      U     #S1; // Select No. 1
      SPB   S1;
      U     #S2; // Select No. 2
      SPB   S2;
      U     #S3; // Select No. 3
      SPB   S3;
      U     #S4; // Select No. 4
      SPB   S4;
      SPA   OFF;

S1:   L     P##ANY1; // Load the Pointer of ANY 1
      L     1; // Wert für Kanalanzeige
      SPA   SAVE;
S2:   L     P##ANY2; // Load the Pointer of ANY 2
      L     2;
      SPA   SAVE;
S3:   L     P##ANY3; // Load the Pointer of ANY 3
      L     3;
      SPA   SAVE;
S4:   L     P##ANY4; // Load the Pointer of ANY 4
      L     4;
      SPA   SAVE;

OFF:  L     P##anyNull; // Create a temporary
      LAR1  ; // NullAny
      L     DW#16#0;
      T     D [AR1,P#0.0];
      T     D [AR1,P#4.0];
      T     W [AR1,P#8.0];

      L     P##anyNull; // Load Pointer to temporary NullAny
      L     0;
      CLR   ; // CLR BIE

SAVE: SAVE  ; // FC-ENO: TRUE IF ChannelSelected
      T     #DSP_CHANNEL; // Anzeige aktiver Kanal
      TAK   ; // P##ANY in AKKU1 zurück
      LAR1  ; // Load the Pointer of the Source Any into AR1
      L     P##RET_VAL; // Load the Pointer of the ReturnValue into
      LAR2  ; // AR2

      L     D [AR1,P#0.0]; // Copy the 10 Bytes of the ANY Pointer to
      T     D [AR2,P#0.0]; // the returned ANY

      L     D [AR1,P#4.0];
      T     D [AR2,P#4.0];

      L     W [AR1,P#8.0];
      T     W [AR2,P#8.0];


END_FUNCTION

FUNCTION "m7b_DB_COMPARE_ByRef" : VOID
TITLE =DB_COMPARE_ByRef
//Vergleicht Anzahl Bytes von 2 Datenbausteinen
//Die Vergleichsroutine arbeitet sehr effektiv, da die Werte nicht als 8-Bit
//sondern als 32-Bit-Werte verglichen werden. Weiterhin müssen die DBs nur einmal
//geöffnet werden, dies erreicht man, indem man einen DB als Global-DB und den
//anderen als Instanz-DB öffnet.
//
//AUTOR: Stefan Maag, Dipl.-Ing. (FH) Elektrotechnik
//DATUM: 10/2010
//INTERNET: www.maagic7.de
//
//AENDERUNGSVERMERKE:
//--------------------------------------------------------------------------------
//DATUM        NAME        AENDERUNG
//--------------------------------------------------------------------------------
//19.10.2010   S.Maag      Basiert auf FC2 CopyDBW_ByRef
//25.10.2010   S.Maag      Wenn keine Einzelbytes mehr zu kopieren sind, dann
//                         darf man nicht zu END springen sondern zu EQ (Daten
//                         gleich)
//--------------------------------------------------------------------------------
//
//HINWEISE:
AUTHOR : 'S.Maag'
FAMILY : Maagic7
VERSION : 0.1


VAR_INPUT
  SOURCE : BLOCK_DB ;
  DEST : BLOCK_DB ;
  SOURCE_BYTE : INT ;
  DEST_Byte : INT ;
  NoOfBytes : INT ;
END_VAR
VAR_TEMP
  QUELL_ADR : DINT ;
  ZIEL_ADR : DINT ;
  AR1 : DINT ;
  LOOPS : INT ;
END_VAR
BEGIN
NETWORK
TITLE =Register sichern
//Adressregister 2 Global- und Instanz DB werden bei CALL-Aufrufen automatisch
//vom System gesichert, bei UC nicht!
      TAR1  #AR1; // Adressregister 1 sichern

NETWORK
TITLE =Adressen für Quell und Ziel-DW als Pointer in Adressregister

      L     #SOURCE_BYTE; // Quelldatenbyte Nr.
      SLD   3; // als Pointer
      L     P#0.0; // 0-Pointer addieren, damit
      +D    ; // Kennungsbits für Pointer gesetzt werden
      LAR1  ; // ins Adressregister 1

      L     #DEST_Byte; // ZieldatenByte-Nr
      SLD   3; // als Pointer
      L     P#0.0;
      +D    ;
      LAR2  ; // ins Adressregister 2
NETWORK
TITLE =Daten vergleichen

      AUF   #SOURCE; // Quell-DB als Global-DB öffnen
      TDB   ; // Global und Instanz-DB tauschen (Quelle wird Instanz-DB)
      AUF   #DEST; // Ziel-DB als Global-DB öffnen

      L     #NoOfBytes; // Anzahl der zu kopierenden Bytes
      L     4; // in Anzahl der 32-Bit-Werte umrechen
      /I    ;
      SPZ   LAST; // Wenn 0 32-Bit Werte, dann weiter mit letzten 3 Bytes
LOOP: T     #LOOPS;
      L     DID [AR1,P#0.0]; // QuellDaten lesen
      L     DBD [AR2,P#0.0]; // VergleichsDaten lesen
      <>D   ; // wenn nicht gleich, dann Ende
      SPB   NEQ;
      +AR1  P#4.0; // Quell-Pointer in AR1 um 4 Bytes erhöhen
      +AR2  P#4.0; // Ziel-Pointer in AR2 um 4 Bytes erhöhen
      L     #LOOPS; // Schleifenzähler wieder in Akku 1 zurück
      LOOP  LOOP; // Schleifenzähler bearbeiten

LAST: L     #NoOfBytes; // nun noch die evtl. letzte 3 Bytes prüfen
      L     2#11; // Anzahl übriger Bytes maskieren
      UW    ; // Anzahl übriger Bytes
      SPZ   EQ; // Wenn 0 dann ENDE
LOP1: T     #LOOPS;
      L     DIB [AR1,P#0.0]; // QuellDaten lesen
      L     DBB [AR2,P#0.0]; // VergleichsDaten lesen
      <>I   ; // wenn nicht gleich, dann Ende
      SPB   NEQ;
      +AR1  P#1.0; // Quell-Pointer in AR1 um 1 Byte erhöhen
      +AR2  P#1.0; // Vergleichs-Pointer in AR2 um 1 Byte erhöhen
      L     #LOOPS; // Schleifenzähler wieder in Akku 1 zurück
      LOOP  LOP1; // Schleifenzähler bearbeiten

EQ:   SET   ; // Daten sind gleich  (equal)
      SAVE  ; // ENO=TRUE
      CLR   ;
      SPA   END;

NEQ:  CLR   ; // Daten sind nicht identisch (not equal)
      SAVE  ; // ENO=FALSE

NETWORK
TITLE =Adressregister 1 wieder herstellen

END:  LAR1  #AR1; // Adressregister 1 wieder herstellen

END_FUNCTION

FUNCTION "m7b_IEC_TIMER_CTRL" : VOID
TITLE =Erweiterte Steuerung von IEC Timern (RESET und 0ms Rüfung)
//IEC-Timer haben im Gegensatz zu den S5-Timern keine RESET-Eingang
//Für RESET eines IEC-Timers muss man diesen mit einer Zeit von 0ms
//aufrufen. (Dies gilt dann als Reset). D.h. IEC-Timer laufen mit
//einer Vorgabe von 0ms nicht an. S5-Timer dagegen gehen bei 0s sofort auf Hi.
//Dieses Verhalten der IEC-Timer führt immer wieder zu Problemen, wenn variable
//Zeitwerte verwendet werden, und 0 eingegeben wird.
//
//Dieser Baustein vor den eigentlichen IEC-Timer geschaltet, ermöglicht gleiches
//Verhalten wie bei S5-Timern.
//
//AUTOR: Stefan Maag, Dipl.-Ing. (FH) Elektrotechnik
//DATUM: 1/2013
//INTERNET: www.maagic7.de
//
//AENDERUNGSVERMERKE:
//--------------------------------------------------------------------------------
//DATUM        NAME        AENDERUNG
//--------------------------------------------------------------------------------
//
//--------------------------------------------------------------------------------
//
//HINWEISE:
AUTHOR : 'S.Maag'
FAMILY : Maagic7
VERSION : 0.1


VAR_INPUT
  IN_TIME : TIME ;	//Vorgabezeit Timer
  RESET : BOOL ;	//RESET Timer
END_VAR
VAR_OUTPUT
  OUT_TIME : TIME ;
END_VAR
BEGIN
NETWORK
TITLE =

      SET   ;
      SAVE  ;
      CLR   ;

NETWORK
TITLE =

      L     T#0MS; // Wenn Reset, dann 0ms als Zeit ausgeben
      U     #RESET; // Ein Aufruf mit T=0ms ist für IEC Timer
      SPB   save; // Ein Reset. Siehe Step7 Dokumentation

      L     T#1MS; // Wenn kein Reset, dann minimale Zeitvorgabe
      L     #IN_TIME; // auf 1ms begrenzen
      <D    ; // sonst läuft Timer nicht los,
      SPB   save; // d.h. Ausgang bleibt Lo, da RESET
      TAK   ;
save: T     #OUT_TIME; // Ausgang Zeit für IEC-Timer

END_FUNCTION

FUNCTION "m7b_IEC_TIMER_WRAPPER" : VOID
TITLE =IEC-TIMER-WRAPPER
//AUTOR: Stefan Maag, Dipl.-Ing. (FH) Elektrotechnik
//DATUM: 8/2013
//INTERNET: www.maagic7.de
//
//AENDERUNGSVERMERKE:
//--------------------------------------------------------------------------------
//DATUM        NAME            AENDERUNG
//--------------------------------------------------------------------------------
//
//--------------------------------------------------------------------------------
//
//HINWEISE:
AUTHOR : 'S.Maag'
FAMILY : Maagic7
VERSION : 0.1


VAR_INPUT
  IN : BOOL ;	//TIMER IN-SIGNAL
  RESET : BOOL ;	//RESET THE TIMER
  cfgDSP_ET_INV : BOOL ;	//Configuration: Display the ET-Time inverted (rest TIME)
  PT : TIME ;	//TIMER PT (TIME)
  ptrTmrInst : POINTER ;	//RELATIVE POINTER TO TIMER INSTANCE: MemoryArea must be in actual instance DB
  TMR_SFB_No : INT ;	//No. of Timer SFB: 3=TP, 4=TON, 5=TOF
END_VAR
VAR_OUTPUT
  ET : TIME ;	//Abgelaufene Zeit
END_VAR
VAR_TEMP
  memAR1 : DWORD ;
  memAR2 : DWORD ;
  TimeIsNull : BOOL ;
END_VAR
BEGIN
NETWORK
TITLE =Save AR1 & AR2

      TAR1  #memAR1; // save AR1, AR2
      TAR2  #memAR2;

NETWORK
TITLE =Load AR2 with Pointer to TIMER-INSTANCE and SET the TIMER
//For the unconditioned call of TIMER SFBs (UC SFB3..5) we have to implement the
//following steps manually:
//1. SET AR2 with correct INSTANCE-POINTER of TIMER
//2. TRANSFER TIMER.VARIABLES into INCTANCE-DATA: (IN and PT)
//
//TIMER_STRUCTURE of SFB 3..5 (TP/TON/TOF) with relative ADDRESS
//   IN      BOOL   0.0  INPUT:  Signal
//   PT      TIME   2.0  INPUT:  TIME
//   Q       BOOL   6.0  OUTPUT: Q
//   ET      TIME   8.0  OUTPUT: ET
//   STATE   BYTE  10.0  static: STATE
//   STIME   TIME  14.0  static: STIME
//   ATIME   TIME  18.0  static: ATIME
//
      L     P##ptrTmrInst; // Load POINTER to ptrTmrInst
      LAR1  ; // in AR1
      L     D [AR1,P#2.0]; // Load relative InstancePointer (Offset 2: don't need DB-No; Byte 0..1)
      UD    DW#16#FFFFFF; // BYTE.BIT-Pointer only: Remove MemoryArea (Speicherbereich)
      +AR2  ; // Instance-DataPointer of TimerInstance [P#Byte.Bit]
      U     #IN; // Timer Startsignal in Instanz eintragen
      =     DIX [AR2,P#0.0]; // [TIMER].IN

      L     #PT; // Zeitwert in TimerInstanz eintragen
      T     DID [AR2,P#2.0]; // [TIMER].PT
      L     L#0; // IF .PT =0 means RESET for IEC-TIMERs
      ==D   ;
      =     #TimeIsNull; // Zeit ist T#0ms  => [TIMER].Q will be FALSE

NETWORK
TITLE =RESET
//// IEC-Timer Reset is done by PT:=0
//IF RESET THEN
//   [TIMER].PT = 0
//ENDIF
      U     #RESET;
      SPBN  ne2;
      L     L#0; // T#0ms means RESET for IEC-TIMERs
      T     DID [AR2,P#2.0]; // [TIMER].PT

ne2:  NOP   0;
NETWORK
TITLE =SELECT TIMER FUNCTION
//SELECT TMR_SFB_No
//  CASE <3 or >5 : ERR
//  CASE 3: SFB3 'TP'
//  CASE 4: SFB4 'TON'
//  CASE 5: SFB5 'TOF'
      L     #TMR_SFB_No;
      SPL   ERR; // >5 (OUT OF RANGE)
      SPA   ERR; // 0
      SPA   ERR; // 1
      SPA   ERR; // 2
      SPA   TP; // 3  SFB3 TP
      SPA   TON; // 4  SFB4 TON
      SPA   TOF; // 5  SFB5 TOF

ERR:  NOP   0; //  *****    E R O R     *****
      CLR   ;
      SAVE  ;
      SPA   END;

TP:   NOP   0; //  ***** M O D E   T P  *****

      UC    "TP"; // unconditioned call for SFB3 'TP'; AR2 has to be loaded with InstanceDataPointer first!

      U     DIX [AR2,P#6.0]; // [TIMER].Q
      SAVE  ;
      CLR   ;
      SPA   END;

TON:  NOP   0; // ***** M O D E   T O N *****

      UC    "TON"; // unconditioned call for SFB4 'TON'; AR2 has to be loaded with InstanceDataPointer first!

      U     #IN; // INPUT SIGNAL for TIMER start
      U     #TimeIsNull;
      O     DIX [AR2,P#6.0]; // [TIMER].Q
      SAVE  ;
      CLR   ;
      SPA   END;

TOF:  NOP   0; // ***** M O D E   T O F *****

      UC    "TOF"; // unconditioned call for SFB5 'TOF'; AR2 has to be loaded with InstanceDataPointer first!

      U     #IN; // INPUT SIGNAL for TIMER start
      U     #TimeIsNull;
      O     DIX [AR2,P#6.0]; // [TIMER].Q
      SAVE  ;
      CLR   ;
      SPA   END;


END:  L     DID [AR2,P#8.0]; // [TIMER].ET   (Laufzeit vom IEC-Timer)
      UN    #cfgDSP_ET_INV; // config Input: Display Time inverted (RestZeit)
      SPB   save;
      L     #PT; // IF inverted THEN
      TAK   ; //    [OUT].ET = PT-TIMER.ET
      -D    ;
save: T     #ET; // [OUT].ET

      LAR1  #memAR1; // restore AR1, AR2
      LAR2  #memAR2;


END_FUNCTION

FUNCTION "m7b_InputControl_REAL" : VOID
TITLE =Input Control for REAL
//Eingabekontrolle für REAL-Werte.
//Begrenzt einen Real-Wert auf vorgegebenen Min/Max Grenzen,
//wobei die Begrenzungsfunktion über Konfigurationseingänge
//zu und abgeschaltet werden kann. So lassen sich z.B. über globale
//Schalter die Eingabebegrenzungen z.B. für Servicezwecke aufheben.
//
//[IN]
//rMIN :         Zulässiger Minimalwert
//rMAX :         Zulässiger Maximalwert
//cfg_LIM_min :  Konfiguration Begrenzung auf Min-Wert aktiv
//cfg_LIM_max :  Konfiguration Begrenzung auf Max-Wert aktiv
//
//[INOUT]
//rVALUE :       Zu prüfender/begrenzender Wert
//
//[OUT]
//MSG_LIM_MAX :  Meldung: Max-Limit überschritten
//MSG_LIM_MIN :  Meldung: Min-Limit unterschritten
//DSP_STATUS :   Status: 0 : o.k. ; 1 : MinLimit; 2 : MaxLimit
//
//AUTOR: Stefan Maag, Dipl.-Ing. (FH) Elektrotechnik
//DATUM: 5/2013
//INTERNET: www.maagic7.de
//
//AENDERUNGSVERMERKE:
//--------------------------------------------------------------------------------
//DATUM        NAME            AENDERUNG
//--------------------------------------------------------------------------------
//
//--------------------------------------------------------------------------------
//
//HINWEISE:
AUTHOR : 'S.Maag'
FAMILY : Maagic7
VERSION : 0.1


VAR_INPUT
  rMIN : REAL ;	//Zulässiger Minimalwert
  rMAX : REAL ;	//Zulässiger Maximalwert
  cfg_LIM_min : BOOL ;	//Konfiguration Begrenzung auf Min-Wert aktiv
  cfg_LIM_max : BOOL ;	//Konfiguration Begrenzung auf Max-Wert aktiv
END_VAR
VAR_OUTPUT
  MSG_LIM_MAX : BOOL ;	//Meldung: Max-Limit überschritten
  MSG_LIM_MIN : BOOL ;	//Meldung: Min-Limit unterschritten
  DSP_STATUS : INT ;	//Status: 0 : o.k. ; 1 : MinLimit; 2 : MaxLimit
END_VAR
VAR_IN_OUT
  rVALUE : REAL ;	//Zu prüfender Wert
END_VAR
BEGIN
NETWORK
TITLE =
//-
      SET   ;
      SAVE  ;
      CLR   ;
NETWORK
TITLE =Begrenzung, wenn aktiv!
//Begrenzen des Wertes, wenn über-/unterschritten
//Begrenzung wird mit den Konfigurationseingängen
//cfg_LIM_min, cfg_LIM_max = HIGH aktiviert.
      L     #rVALUE; // Sollwert
      L     #rMIN; // minimal Wert
      <R    ;
      U     #cfg_LIM_min;
      SPB   LIM; // Limitierung wenn VALUE < MIN
      TAK   ; // VALUE wieder in Akku 1
      L     #rMAX; // Maximalwert
      >R    ;
      U     #cfg_LIM_max;
      SPB   LIM; // Limitierung wenn VALUE > MAX

      SPA   ne;
      CLR   ; // VKE löschen, da keine Begrenzung erfolgte
      SAVE  ; // BIE-Bit = 0, da Wert im Bereich war; ="Keine Begrenzung"
      BEA   ;

LIM:  T     #rVALUE; // max.Wert als Sollwert ausgeben

ne:   NOP   0;

NETWORK
TITLE =Meldeausgänge Limit überschritten
//-
      L     #rVALUE;
      L     #rMAX; // minmal zulässiger Wert
      >R    ; // falls MIN > VALUE
      =     #MSG_LIM_MAX;

      L     #rVALUE;
      L     #rMIN; // minmal zulässiger Wert
      <R    ; // falls MIN > VALUE
      =     #MSG_LIM_MIN;

NETWORK
TITLE =STATUS
//0 : o.k., keine Begreunzung aktiv
//1 : Begrenzung min
//2 : Begrenzung max
      L     1;
      U     #MSG_LIM_MIN;
      SPB   save;

      L     2;
      U     #MSG_LIM_MAX;
      SPB   save;

      L     0;
save: T     #DSP_STATUS;
END_FUNCTION

FUNCTION "m7b_InputControl_DINT" : VOID
TITLE =Input Control for DINT
//Eingabekontrolle für DINT-Werte.
//Begrenzt einen Real-Wert auf vorgegebenen Min/Max Grenzen,
//wobei die Begrenzungsfunktion über Konfigurationseingänge
//zu und abgeschaltet werden kann. So lassen sich z.B. über globale
//Schalter die Eingabebegrenzungen z.B. für Servicezwecke aufheben.
//
//[IN]
//dMIN :         Zulässiger Minimalwert
//dMAX :         Zulässiger Maximalwert
//cfg_LIM_min :  Konfiguration Begrenzung auf Min-Wert aktiv
//cfg_LIM_max :  Konfiguration Begrenzung auf Max-Wert aktiv
//
//[INOUT]
//dVALUE :       Zu prüfender/begrenzender Wert
//
//[OUT]
//MSG_LIM_MAX :  Meldung: Max-Limit überschritten
//MSG_LIM_MIN :  Meldung: Min-Limit unterschritten
//DSP_STATUS :   Status: 0 : o.k. ; 1 : MinLimit; 2 : MaxLimit
//
//AUTOR: Stefan Maag, Dipl.-Ing. (FH) Elektrotechnik
//DATUM: 10/2017
//INTERNET: www.maagic7.de
//
//AENDERUNGSVERMERKE:
//--------------------------------------------------------------------------------
//DATUM        NAME            AENDERUNG
//--------------------------------------------------------------------------------
//31.10.2017   S.Maag         Entstand aus FC252 InputControl_REAL
//--------------------------------------------------------------------------------
//
//HINWEISE:
AUTHOR : 'S.Maag'
FAMILY : Maagic7
VERSION : 0.1


VAR_INPUT
  dMIN : DINT ;	//Zulässiger Minimalwert
  dMAX : DINT ;	//Zulässiger Maximalwert
  cfg_LIM_min : BOOL ;	//Konfiguration Begrenzung auf Min-Wert aktiv
  cfg_LIM_max : BOOL ;	//Konfiguration Begrenzung auf Max-Wert aktiv
END_VAR
VAR_OUTPUT
  MSG_LIM_MAX : BOOL ;	//Meldung: Max-Limit überschritten
  MSG_LIM_MIN : BOOL ;	//Meldung: Min-Limit unterschritten
  DSP_STATUS : INT ;	//Status: 0 : o.k. ; 1 : MinLimit; 2 : MaxLimit
END_VAR
VAR_IN_OUT
  dVALUE : DINT ;	//Zu prüfender Wert
END_VAR
BEGIN
NETWORK
TITLE =
//-
      SET   ;
      SAVE  ;
      CLR   ;
NETWORK
TITLE =Begrenzung, wenn aktiv!
//Begrenzen des Wertes, wenn über-/unterschritten
//Begrenzung wird mit den Konfigurationseingängen
//cfg_LIM_min, cfg_LIM_max = HIGH aktiviert.
      L     #dVALUE; // Sollwert
      L     #dMIN; // minimal Wert
      <D    ;
      U     #cfg_LIM_min;
      SPB   LIM; // Limitierung wenn VALUE < MIN
      TAK   ; // VALUE wieder in Akku 1
      L     #dMAX; // Maximalwert
      >D    ;
      U     #cfg_LIM_max;
      SPB   LIM; // Limitierung wenn VALUE > MAX

      SPA   ne;
      CLR   ; // VKE löschen, da keine Begrenzung erfolgte
      SAVE  ; // BIE-Bit = 0, da Wert im Bereich war; ="Keine Begrenzung"
      BEA   ;

LIM:  T     #dVALUE; // max.Wert als Sollwert ausgeben

ne:   NOP   0;

NETWORK
TITLE =Meldeausgänge Limit überschritten
//-
      L     #dVALUE;
      L     #dMAX; // minmal zulässiger Wert
      >D    ; // falls MIN > VALUE
      =     #MSG_LIM_MAX;

      L     #dVALUE;
      L     #dMIN; // minmal zulässiger Wert
      <D    ; // falls MIN > VALUE
      =     #MSG_LIM_MIN;

NETWORK
TITLE =STATUS
//0 : o.k., keine Begreunzung aktiv
//1 : Begrenzung min
//2 : Begrenzung max
      L     1;
      U     #MSG_LIM_MIN;
      SPB   save;

      L     2;
      U     #MSG_LIM_MAX;
      SPB   save;

      L     0;
save: T     #DSP_STATUS;
END_FUNCTION

FUNCTION "m7b_BetriebsStunden" : VOID
TITLE =Betriebsstunden erfassen
//pro Bausteinaufruf wird eine bestimmte Anzahl von Sekunden addiert.
//Diesen Baustein mit einem Referenztakt (Timer OB, oder Flanke von Taktmerker
//aufrufen)
//
//AUTOR: Stefan Maag, Dipl.-Ing. (FH) Elektrotechnik
//DATUM: 8/2013
//INTERNET: www.maagic7.de
//
//AENDERUNGSVERMERKE:
//--------------------------------------------------------------------------------
//DATUM        NAME            AENDERUNG
//--------------------------------------------------------------------------------
//04.12.2013   S.Maag      Bei Count-Aufruf über EN, funktionieren Impulsausgänge
//                         nicht, deswegen Count-Eingang eingeführt
//--------------------------------------------------------------------------------
//
//HINWEISE:
AUTHOR : 'S.Maag'
FAMILY : Maagic7
VERSION : 0.1


VAR_INPUT
  COUNT : BOOL ;	//Eingang zählen
  RESET : BOOL ;	//Tageszähler löschen
  SEC_ADD : INT ;
END_VAR
VAR_OUTPUT
  IMP_MIN : BOOL ;
  IMP_H : BOOL ;
END_VAR
VAR_IN_OUT
  sec : INT ;
  min : INT ;
  h : DINT ;	//Stunden
END_VAR
BEGIN
NETWORK
TITLE =

      SET   ;
      SAVE  ;
      R     #IMP_MIN;
      R     #IMP_H;
      CLR   ;

      UN    #RESET;
      SPB   cnt;
      L     0;
      T     #sec;
      T     #min;
      T     #h;
      BEA   ;

cnt:  UN    #COUNT;
      BEB   ;

      L     #sec;
      L     #SEC_ADD;
      +I    ;
      T     #sec;
      L     60;
      <I    ;
      BEB   ;

      S     #IMP_MIN;

      L     #sec;
      +     -60;
      T     #sec;

      L     #min;
      +     1;
      T     #min;

      L     60;
      <I    ;
      BEB   ;

      S     #IMP_H;

      L     #min;
      +     -60;
      T     #min;

      L     #h;
      +     1;
      T     #h;
      L     0; // Überlauf prüfen, Stunden müssen >=0 sein
      >=D   ; // wenn nicht, dann auf 0 setzten
      BEB   ;
      T     #h;
END_FUNCTION

FUNCTION "m7b_DeltaTime" : VOID
TITLE =DeltaTime : Zeitdifferenz zwischen 2 Impulsen
//Ermittelt den Abstand zwischen 2 Impulsen.
//In io_DeltaTime wird der Abstand des letzten Impulses gespeichert.
//DSP_ActTimDiff zeigt die seit letztem Impuls aktuell vergangene Zeit
//MAX_timDiff = MAX(io_DeltaTime, DSP_TimeDiffAkt)
//
//
//AUTOR: Stefan Maag, Dipl.-Ing. (FH) Elektrotechnik
//DATUM: 11/2013
//INTERNET: www.maagic7.de
//
//AENDERUNGSVERMERKE:
//--------------------------------------------------------------------------------
//DATUM        NAME        AENDERUNG
//--------------------------------------------------------------------------------
//04/09/2017   S.Maag      RESET Eingang + einfrieren 1sec vor max Differenz
//
//16/01/2014   S.Maag      ENO=TRUE
//
//03/12/2013   S.Maag      SFC64 TimeTick Zeitdifferenz korrigiert
//                         da 31Bit, Fehler bei Überlauf.
//                         jetzt Differenzber. mit FC256 "ABS_DIFF_S7SysTime"
//--------------------------------------------------------------------------------
//
//HINWEISE:
AUTHOR : 'S.Maag'
FAMILY : Maagic7
VERSION : 0.1


VAR_INPUT
  FP_Signal : BOOL ;	//Flanke Signal
  RESET : BOOL ;
END_VAR
VAR_OUTPUT
  DSP_ActTimeDiff : TIME ;	//Anzeige aktuelle Zeitdifferenz seit letztem Ereignis
  MAX_timDiff : TIME ;	//Max(timDiff, io_DeltaTime)
END_VAR
VAR_IN_OUT
  memTime : TIME ;
  io_DeltaTime : TIME ;
END_VAR
VAR_TEMP
  SysTimer : TIME ;
END_VAR
BEGIN
NETWORK
TITLE =

      SET   ;
      SAVE  ;
      CLR   ;

NETWORK
TITLE =
//31Bit = 7F FF FF FF = 2147483647 - 1000ms = 2147482647 ms
//1sec vor Ablauf der max Differenz den Differenzwert einfrieren bis neuer Impuls
//kommt.
//Dies verhindert Überlauf der Zeitdifferenz uns somit eine Rückfall der
//Differenzzeit auf 0 ohne neuen Impuls
      UN    #RESET;
      SPB   do;

      L     T#0MS;
      T     #DSP_ActTimeDiff;
      T     #MAX_timDiff;
      SPA   ne2;

do:   NOP   0;
      CALL "TIME_TCK" (
           RET_VAL                  := #SysTimer);

      L     #DSP_ActTimeDiff; // Wenn max. Zeitdifferenz erreicht,
      L     L#2147482647; // dann Wert einfrieren und erst
      >=D   ; // nach neuem Impuls weiter
      SPB   ne2; // dadurch wird ein überlauf verhindert

      L     #SysTimer;
      L     #memTime;
      UC    "m7b_ABS_DIFF_S7SysTime"; // Absolute Zeitdifferenz S7-SystemTimer 31Bit
      T     #DSP_ActTimeDiff;
      L     #io_DeltaTime;
      UC    FC    21;
      T     #MAX_timDiff;
ne2:  NOP   0;
NETWORK
TITLE =Zeit Ereignis

      UN    #FP_Signal;
      SPB   ne3;

      L     #DSP_ActTimeDiff;
      T     #io_DeltaTime;

      L     L#0;
      T     #DSP_ActTimeDiff;

      L     #SysTimer;
      T     #memTime;

ne3:  NOP   0;
NETWORK
TITLE =



END_FUNCTION

FUNCTION "m7b_CNT_UpDwn_IMP_MM.SS" : VOID
TITLE =Zählt Impulse im Minuten.Sekunden Format (MM.SS) - DINT
//Bei jedem Aufruf Zählt diese Funktion einen Impuls weiter. Die Wertedarstellung
//erfolgt im Minuten.Sekunden-Format MM.SS. Es wird also alle 60 Impulse ein
//Überlauf auf MM erzeugt. Dieser Baustein eignet sich zum Erfassen von z.B.
//Behälter Füll- und Entleerzeiten, wenn er mit einer Sekundenflanke aufgerufen
//wird. Am besten Flanke des Systemtaktmerkers 1 sec verwenden.
//
//Der FC-ENO Ausgang ist immer dan HIGH, wenn Zeit > 0
//
//AUTOR: Stefan Maag, Dipl.-Ing. (FH) Elektrotechnik
//DATUM: 5/2005
//
//AENDERUNGSVERMERKE:
//--------------------------------------------------------------------------------
//DATUM        NAME            AENDERUNG
//--------------------------------------------------------------------------------
//25.06.2019   S.Maag     COUNT_UP / COUNT_DOWN
//                        Ausgang d_mmss als I/O, somit muss nur bei Änderung
//                        neu berechnet werden.
//                        ENO = (Time > 0) d.h. ENO=FALSE, wenn Zeit = 0
//                        Wird für Rückwärtszählung benötigt!
//
//14.08.2013   S.Maag     Ausgang MM.SS hinzugefügt so dass im IO mem_dIMP die
//                        gezählten Impulse stehen und nicht mehr MM.SS
//--------------------------------------------------------------------------------
//
//HINWEISE:
AUTHOR : 'S.Maag'
FAMILY : Maagic7
VERSION : 0.1


VAR_INPUT
  COUNT_UP : BOOL ;	//Signal for counting up
  COUNT_DWN : BOOL ;	//Signal for counting down
  SET : BOOL ;	//Set to VALUE_SET
  VALUE_SET_mmss : DINT ;	//Value [mm:ss] to set
END_VAR
VAR_IN_OUT
  io_dIMP : DINT ;	//Memory for impulses [sec]
  io_d_mmss : DINT ;	//Memory [mm:ss] format
END_VAR
VAR_TEMP
  SS : INT ;
  MM : DINT ;
END_VAR
BEGIN
NETWORK
TITLE =



NETWORK
TITLE =SET

      UN    #SET;
      SPB   NE1;

      L     #VALUE_SET_mmss;
      L     L#100;
      MOD   ; // Sekundenanteil 0..99
      T     #SS; // =Divisionsrest = Sekunden

      L     #VALUE_SET_mmss;
      L     L#100; // Minutenanteil
      /D    ;
      T     #MM; // Rückrechnung auf Sekunden
      L     L#60; // damit werden automatisch
      *D    ; // Sekundenanteile von 60..99
      L     #SS; // auf eine zusätzliche Minute
      +D    ; // umgerechnet
      T     #io_dIMP;
      SPA   END;
NE1:  NOP   0;
NETWORK
TITLE =Impulse Zählen [mm:ss]
//
//
      U     #COUNT_UP;
      SPB   up;
      U     #COUNT_DWN;
      SPB   dwn;

      SPA   END;

up:   L     #io_dIMP;
      +     L#1;
      SPA   chk;
dwn:  L     #io_dIMP;
      +     L#-1;
chk:  L     L#0; // wenn <0, dann 0
      <D    ; // das begrenzt sowohl bei down
      SPB   save; // als auch Überläufe bei UP auf negative Zeit
      TAK   ;
save: T     #io_dIMP;
      L     L#60; // Sekunden pro Minute
      /D    ;
      T     #MM; // Minuten

      L     #io_dIMP;
      L     L#60; // Sekunden pro Minute
      MOD   ; // Restwerdivision: Rest sec
      T     #SS; // =Divisionsrest = Sekunden

      L     #MM; // Minuten*100
      L     L#100;
      *D    ;
      L     #SS;
      +D    ;
      T     #io_d_mmss; // Wert in MM.SS

END:  L     #io_dIMP;
      L     L#0;
      >D    ;
      SAVE  ;
      CLR   ;

END_FUNCTION

FUNCTION "m7b_CNT_Up" : VOID
TITLE =Simple up counter
//AUTOR: Stefan Maag, Dipl.-Ing. (FH) Elektrotechnik
//DATUM: 4/2020
//
//AENDERUNGSVERMERKE:
//--------------------------------------------------------------------------------
//DATUM        NAME        AENDERUNG
//--------------------------------------------------------------------------------
//
//--------------------------------------------------------------------------------
//
//HINWEISE:
AUTHOR : 'S.Maag'
FAMILY : Maagic7
VERSION : 0.1


VAR_INPUT
  xCnt : BOOL ;	//Count: Hi is continous counting
  xReset : BOOL ;	//Reset counter to 0
END_VAR
VAR_IN_OUT
  io_dCNT : DINT ;	//io Counter value
END_VAR
BEGIN
NETWORK
TITLE =

NETWORK
TITLE =count

      U     #xCnt;
      SPBNB _001;
      L     #io_dCNT;
      L     L#1;
      +D    ;
      T     #io_dCNT;
_001: NOP   0;
NETWORK
TITLE =Reset

      U     #xReset;
      SPBNB _002;
      L     0;
      T     #io_dCNT;
_002: NOP   0;
NETWORK
TITLE =

      SET   ;
      SAVE  ;
      CLR   ;

END_FUNCTION

FUNCTION "m7b_CNT_UpDwn_Limit" : VOID
TITLE =Couter Up Down with Limit
//Counter Up Down with liumit for up and down
//If the limit is reached the counter stops counting.
//32-Bit DINT: -2147483648 to +2147483647
//
//How to use this counter:
//
//- As Timer if you count with the SystemClockFlags. In contrast to IEC Timer
//  this one is easy to pause!
//
//- As standard counter because IEC counters only use 16-Bit values
//
//
//AUTOR: Stefan Maag, Dipl.-Ing. (FH) Elektrotechnik
//DATUM: 4/2020
//
//AENDERUNGSVERMERKE:
//--------------------------------------------------------------------------------
//DATUM        NAME        AENDERUNG
//--------------------------------------------------------------------------------
//24.03.2021   S.Maag      FB wasn't ready programmed! Finished!
//                         Added seperate limit for down!
//                         Added seperate Output signals for Limit up/down reached
//                         Changend cfgUpDwn to cfgDwnUp (!more logical)
//--------------------------------------------------------------------------------
//
//HINWEISE:
AUTHOR : 'S.Maag'
FAMILY : Maagic7
VERSION : 0.1


VAR_INPUT
  xCntUp : BOOL ;	//1: count up; 0: do nothing
  xCntDwn : BOOL ;	//1: count dwon; 0: do nothing
  xSET : BOOL ;	//Set counter to SetVal
  dSetVal : DINT ;	//Set value
  dCntVal : DINT ;	//io_dCount +/- dCntVal
  dLimitUp : DINT ;	//Limit up (-2147483648..2147483647)
  dLimitDwn : DINT ;	//Limit down (-2147483648..2147483647)
END_VAR
VAR_OUTPUT
  Q_LIM_UP : BOOL ;
  Q_LIM_DWN : BOOL ;
END_VAR
VAR_IN_OUT
  io_dCNT : DINT ;	//io Zählerwert
END_VAR
BEGIN
NETWORK
TITLE =



NETWORK
TITLE =Set the counter to SetVal
//IF xSET THEN io_dCNT := dSetVal; END_IF;
      U     #xSET;
      SPBNB _001;
      L     #dSetVal;
      T     #io_dCNT;
_001: NOP   0;
NETWORK
TITLE =Count up
//IF xCntUp THEN
//   io_dCnt := io_dCnt + dCntVal;
//   IF OVERFLOW OR (iodCnt > dLimitUp) THEN
//      iodCnt := dLimitUp;
//   END_IF;
//END_IF;
//
      U     #xCntUp; // IF CntUp
      SPBN  NE2;

      L     #io_dCNT; // Counter value
      L     #dCntVal; // Value to count
      +D    ;
      L     #dLimitUp; // Counter upper limit
      U     OV; // Overflow Bit
      O     ;
      >D    ; // io_dCNT + dCntVal > LimitUp
      SPB   SUp; // save CntUp => save Limit
      TAK   ; // io_dCNT + dCntVal => Akku1
SUp:  T     #io_dCNT; // save the new counter value
NE2:  NOP   0;

NETWORK
TITLE =Count down
//IF xCntDwn THEN
//   io_dCnt := io_dCnt - dCntVal;
//   IF OVERFLOW OR (iodCnt < dLimitDwn) THEN
//      iodCnt := dLimitDwn;
//   END_IF;
//END_IF;
      U     #xCntDwn; // IF CntDwn
      SPBN  NE3;

      L     #io_dCNT; // Counter value
      L     #dCntVal; // Value to count
      -D    ;
      L     #dLimitDwn; // Counter lower limit
      U     OV; // Overflow Bit
      O     ;
      <D    ; // io_dCNT - dCntVal < LimitDwn
      SPB   SDwn; // save CntUp => save Limit
      TAK   ; // io_dCNT - dCntVal => Akku1
SDwn: T     #io_dCNT; // save the new counter value
NE3:  NOP   0;

NETWORK
TITLE =Limit up reached ?
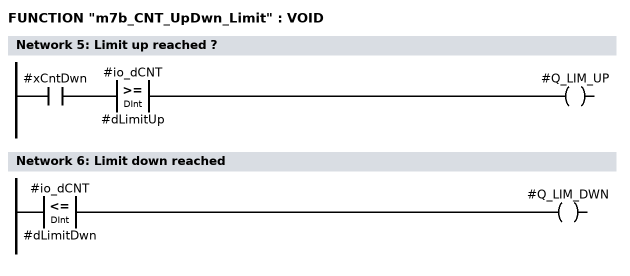

      U     #xCntDwn;
      U(    ;
      L     #io_dCNT;
      L     #dLimitUp;
      >=D   ;
      )     ;
      =     #Q_LIM_UP;
NETWORK
TITLE =Limit down reached

      L     #io_dCNT;
      L     #dLimitDwn;
      <=D   ;
      =     #Q_LIM_DWN;
NETWORK
TITLE =

      SET   ;
      SAVE  ;

END_FUNCTION

FUNCTION "m7b_mmss_Overflow" : VOID
TITLE =Check and correct Overflow of hh:mm or mm:ss variables
//mmss_Overflow:
//Check and correct the overflow of variables with time values in the [hh:mm] or
//[mm:ss] Format.
//
//Example:
//Value = 259  ;  2h 59m -> correct, nothing to do
//Value = 260  ;  2h 60m -> correct to 3h 00m by adding 40 -> Value = 300
//Value = 265  ;  2h 65m -> correct to 3h 05m by adding 40 -> Value = 305
//
//FC_ENO = TRUE if there was an overflow
//
//AUTOR: Stefan Maag, Dipl.-Ing. (FH) Elektrotechnik
//DATUM: 9/2019
//
//AENDERUNGSVERMERKE:
//--------------------------------------------------------------------------------
//DATUM        NAME            AENDERUNG
//-------------------------------------------------------------------------------
AUTHOR : 'S.Maag'
FAMILY : Maagic7
VERSION : 0.1


VAR_IN_OUT
  io_d_hhmm_mmss : DINT ;	//Input value in hh:mm or mm:ss
END_VAR
BEGIN
NETWORK
TITLE =

      L     #io_d_hhmm_mmss;
      L     L#100; // select lower 2 digits
      MOD   ;
      L     L#60; // full mm or ss
      >=D   ;
      SPBB  OFlw; // Jump if VKE=1 and Save VKE to BIE (Overflow)
      BEA   ;

OFlw: L     #io_d_hhmm_mmss; // we must count 58,59,100 (=add 40 if >=60)
      +     L#40; // Add the correct value for overflow
      T     #io_d_hhmm_mmss; //

END_FUNCTION

FUNCTION "m7b_ImpulsTeiler" : VOID
TITLE =Impulsteiler
//AUTOR: Stefan Maag, Dipl.-Ing. (FH) Elektrotechnik
//DATUM: 12/2015
//
//AENDERUNGSVERMERKE:
//--------------------------------------------------------------------------------
//DATUM        NAME            AENDERUNG
//--------------------------------------------------------------------------------
//
//--------------------------------------------------------------------------------
//
//HINWEISE: In Library aufgenommen 05/2019
AUTHOR : 'S.Maag'
FAMILY : Maagic7
VERSION : 0.1


VAR_INPUT
  Impuls : BOOL ;
  dTeilung : DINT ;	//Impulsteilung: alle x Impulse am Eingang 1x Ausgang
END_VAR
VAR_OUTPUT
  Q : BOOL ;
END_VAR
VAR_IN_OUT
  memDI : DINT ;
END_VAR
VAR_TEMP
  HM_Q : BOOL ;
END_VAR
BEGIN
NETWORK
TITLE =



NETWORK
TITLE =



      U     #Impuls;
      SPBNB _001;
      L     #memDI;
      L     L#1;
      +D    ;
      T     #memDI;
_001: NOP   0;
NETWORK
TITLE =

      L     #memDI;
      L     #dTeilung;
      >=D   ;
      =     #Q;
      =     #HM_Q;
NETWORK
TITLE =

      U     #HM_Q;
      SPBNB _002;
      L     0;
      T     #memDI;
      SET   ;
      SAVE  ;
      CLR   ;
_002: U     BIE;
      SAVE  ;
END_FUNCTION

FUNCTION "m7h_Check4xInput_REAL" : VOID
TITLE =4 Schwellen prüfen: auf- oder absteigend
//Plausiblitätsprüfung von Auf- oder Absteigenden Grenzwerten.
//z.B. Füllstandsschwellen von Behältern. (min darf nicht > max sein)
//[IN]
//cfg_Limit_ON : FALSE : keine Begrenzung der Eingabewerte
//               TRUE  : Begrenzung der Eingabewerte Fehleingaben
//                       werden nicht zugelassen.
//
//cfg_ASC_DESC : FALSE : aufsteigen S1<S2<S3<S4
//               TRUE  : absteigend S1>S2>S3>S4
//
//AUTOR: Stefan Maag, Dipl.-Ing. (FH) Elektrotechnik
//DATUM: 07/2012
//
//AENDERUNGSVERMERKE:
//--------------------------------------------------------------------------------
//DATUM        NAME       AENDERUNG
//--------------------------------------------------------------------------------
//14.03.2020   S.Maag     in Library aufgenommen und Code optimiert
//                        (FLAGs direkt aus Lokaldatenbyte kopiert statt über
//                         FC1 zusammengesetzt)
//
//--------------------------------------------------------------------------------
//
//HINWEISE:
AUTHOR : 'S.Maag'
FAMILY : Maagic7
VERSION : 0.1


VAR_INPUT
  cfg_Limit_ON : BOOL ;	//Schaltet die Begrenzung Ein, sonst nur Anzeige, wenn Schwelle inkonsistent
  cfg_ASC_DESC : BOOL ;	//FALSE: 'ASC' aufsteigende Werte S2>S1 / TRUE: 'DESC' absteigende Werte S2<S1
END_VAR
VAR_OUTPUT
  FLAGs_ok : BYTE ;
END_VAR
VAR_IN_OUT
  S1 : REAL ;
  S2 : REAL ;
  S3 : REAL ;
  S4 : REAL ;
END_VAR
VAR_TEMP
  S1_ok : BOOL ;
  S2_ok : BOOL ;
  S3_ok : BOOL ;
  S4_ok : BOOL ;
END_VAR
BEGIN
NETWORK
TITLE =



NETWORK
TITLE =Lokaldatnwort 0 löschen
//wird benötigt, da S1_0k .. S4_ok als FLAGs ausgegeben wird.
//Damit keine Signale in den Leerbits sind, muss zuvor gelöscht werden.
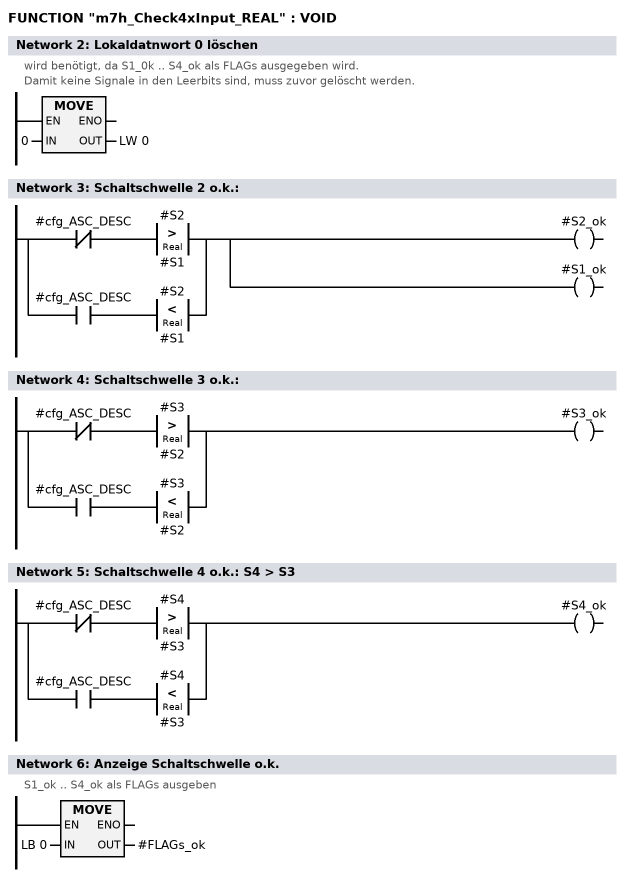
      L     0;
      T     LW     0;
      NOP   0;
NETWORK
TITLE =Schaltschwelle 2 o.k.:

      UN    #cfg_ASC_DESC;
      U(    ;
      L     #S2;
      L     #S1;
      >R    ;
      )     ;
      O     ;
      U     #cfg_ASC_DESC;
      U(    ;
      L     #S2;
      L     #S1;
      <R    ;
      )     ;
      =     #S2_ok;
      =     #S1_ok;
NETWORK
TITLE =Schaltschwelle 3 o.k.:

      UN    #cfg_ASC_DESC;
      U(    ;
      L     #S3;
      L     #S2;
      >R    ;
      )     ;
      O     ;
      U     #cfg_ASC_DESC;
      U(    ;
      L     #S3;
      L     #S2;
      <R    ;
      )     ;
      =     #S3_ok;
NETWORK
TITLE =Schaltschwelle 4 o.k.: S4 > S3

      UN    #cfg_ASC_DESC;
      U(    ;
      L     #S4;
      L     #S3;
      >R    ;
      )     ;
      O     ;
      U     #cfg_ASC_DESC;
      U(    ;
      L     #S4;
      L     #S3;
      <R    ;
      )     ;
      =     #S4_ok;
NETWORK
TITLE =Anzeige Schaltschwelle o.k.
//S1_ok .. S4_ok als FLAGs ausgeben
      L     LB     0;
      T     #FLAGs_ok;
      NOP   0;
NETWORK
TITLE =

      UN    #cfg_Limit_ON;
      BEB   ;

      U     #S4_ok;
      SPB   lim3;

      L     #S3;
      T     #S4;

lim3: U     #S3_ok;
      SPB   lim2;

      L     #S2;
      T     #S3;

lim2: U     #S2_ok;
      SPB   END;

      L     #S1;
      T     #S2;

END:  NOP   0;
NETWORK
TITLE =

      SET   ;
      SAVE  ;


END_FUNCTION

FUNCTION "m7h_Check2xInput_REAL" : VOID
TITLE =2 Schwellen prüfen: auf- oder absteigend
//Plausiblitätsprüfung von Auf- oder Absteigenden Grenzwerten.
//z.B. Füllstandsschwellen von Behältern. (min darf nicht > max sein)
//[IN]
//cfg_Limit_ON : FALSE : keine Begrenzung der Eingabewerte
//               TRUE  : Begrenzung der Eingabewerte Fehleingaben
//                       werden nicht zugelassen.
//
//cfg_ASC_DESC : FALSE : aufsteigen S1<S2
//               TRUE  : absteigend S1>S2
//
//
//AUTOR: Stefan Maag, Dipl.-Ing. (FH) Elektrotechnik
//DATUM: 11/2016
//
//AENDERUNGSVERMERKE:
//--------------------------------------------------------------------------------
//DATUM        NAME       AENDERUNG
//--------------------------------------------------------------------------------
//14.03.2020   S.Maag     in Library aufgenommen und Code optimiert
//                        (FLAGs direkt aus Lokaldatenbyte kopiert statt über
//                         FC1 zusammengesetzt)
//
//--------------------------------------------------------------------------------
//
//HINWEISE: entsand aus FC346 4 Schwellen prüfen
AUTHOR : 'S.Maag'
FAMILY : Maagic7
VERSION : 0.1


VAR_INPUT
  cfg_Limit_ON : BOOL ;	//Schaltet die Begrenzung Ein, sonst nur Anzeige, wenn Schwelle inkonsistent
  cfg_ASC_DESC : BOOL ;	//FALSE: 'ASC' aufsteigende Werte S2>S1 / TRUE: 'DESC' absteigende Werte S2<S1
END_VAR
VAR_OUTPUT
  FLAGs_ok : BYTE ;
END_VAR
VAR_IN_OUT
  S1 : REAL ;
  S2 : REAL ;
END_VAR
VAR_TEMP
  S1_ok : BOOL ;
  S2_ok : BOOL ;
  S3_ok : BOOL ;
  S4_ok : BOOL ;
END_VAR
BEGIN
NETWORK
TITLE =



NETWORK
TITLE =Lokaldatnwort 0 löschen
//wird benötigt, da S1_0k .. S4_ok als FLAGs ausgegeben wird.
//Damit keine Signale in den Leerbits sind, muss zuvor gelöscht werden.
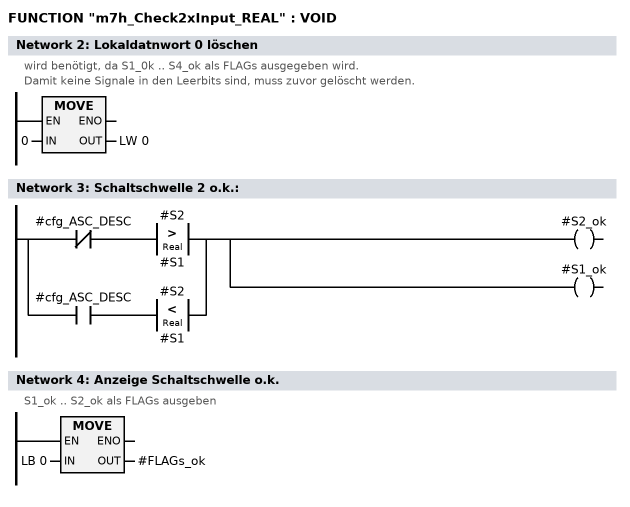
      L     0;
      T     LW     0;
      NOP   0;
NETWORK
TITLE =Schaltschwelle 2 o.k.:

      UN    #cfg_ASC_DESC;
      U(    ;
      L     #S2;
      L     #S1;
      >R    ;
      )     ;
      O     ;
      U     #cfg_ASC_DESC;
      U(    ;
      L     #S2;
      L     #S1;
      <R    ;
      )     ;
      =     #S2_ok;
      =     #S1_ok;
NETWORK
TITLE =Anzeige Schaltschwelle o.k.
//S1_ok .. S2_ok als FLAGs ausgeben
      L     LB     0;
      T     #FLAGs_ok;
      NOP   0;
NETWORK
TITLE =

      UN    #cfg_Limit_ON;
      BEB   ;

      U     #S2_ok;
      SPB   END;

      L     #S1;
      T     #S2;

END:  NOP   0;
NETWORK
TITLE =

      SET   ;
      SAVE  ;


END_FUNCTION

FUNCTION "m7b_MinMax_ERROR_REAL" : VOID
TITLE =Wert ausserhalb Min..Max Bereich und erzeugt Fehlermeldung
//Prüft ob der IST-Wert zwischen MIN & MAX liegt und erzeugt speichernde
//Fehlermeldung.
//
//Verwendung: Fehlerüberwachung von Analogsensoren
//
//AUTOR: Stefan Maag, Dipl.-Ing. (FH) Elektrotechnik
//DATUM: 11/2012
//
//AENDERUNGSVERMERKE:
//--------------------------------------------------------------------------------
//DATUM        NAME            AENDERUNG
//--------------------------------------------------------------------------------
//29.07.2013   S.Maag          Ausgang Statusanzeige hinzugefügt
//--------------------------------------------------------------------------------
//
//HINWEISE: Entstand aus FB38 MinMaxOK_REAL, in Library aufgenommen 03/2020
//          als FC338 beibehalten
AUTHOR : 'S.Maag'
FAMILY : Maagic7
VERSION : 2.0


VAR_INPUT
  VALUE : REAL ;	//Zu prüfender Wert
  MIN : REAL ;	//Zulässiger Minimalwert
  MAX : REAL ;	//Zulässiger Maximalwert
  RESET : BOOL ;
END_VAR
VAR_OUTPUT
  DSP_STATUS : INT ;	//STATUS: 0=o.k.; 1=warn; 2=Fehler
END_VAR
VAR_IN_OUT
  ERR : BOOL ;	//Wert im Toleranzbereich
END_VAR
BEGIN
NETWORK
TITLE =

      L     #MIN; // minmal zulässiger Wert
      L     #VALUE;
      >R    ; // falls MIN > VALUE
      SPB   err; // dann nicht ok
      L     #MAX;
      >R    ; // falls VALUE > MAX
      SPB   err; // dann nicht ok

      U     #RESET;
      R     #ERR; // sonst ok
      SPA   END;

err:  S     #ERR; // Wert nicht ok

END:  UN    #ERR;
      SAVE  ;

NETWORK
TITLE =Statusanzeige
//0 := o.k.
//1 := Warnung
//2 := Fehler
      L     2;
      U     #ERR; // Fehler
      SPB   save;
      L     1;
      CLR   ; // Warnung
      SPB   save;
      L     0; // o.k.
save: T     #DSP_STATUS;
END_FUNCTION

FUNCTION "m7b_HYS_to_MinMax_REAL" : VOID
TITLE =Sollwert mit Hysterese auf min/max umrechnen [REAL]
//AUTOR: Stefan Maag, Dipl.-Ing. (FH) Elektrotechnik
//DATUM: 09/2011
//
//AENDERUNGSVERMERKE:
//--------------------------------------------------------------------------------
//DATUM        NAME            AENDERUNG
//--------------------------------------------------------------------------------
//
//--------------------------------------------------------------------------------
//
//HINWEISE: In Library aufgenommen 03/2020
AUTHOR : 'S.Maag'
FAMILY : Maagic7
VERSION : 0.1


VAR_INPUT
  rSOLL : REAL ;
  rHYS : REAL ;
  cfgFullHys : BOOL ;	//0:= Soll +- Hys/2 ; 1:= Soll +- Hys
END_VAR
VAR_OUTPUT
  rMin : REAL ;
  rMax : REAL ;
END_VAR
VAR_TEMP
  tmpHys : REAL ;
END_VAR
BEGIN
NETWORK
TITLE =

      SET   ;
      SAVE  ;
      CLR   ;

NETWORK
TITLE =Konfiguration halbe oder volle Hysteres
//#cfgFullHys: 0:= Soll +- Hys/2
//             1:= Soll +- Hys
      L     #rHYS;
      U     #cfgFullHys;
      SPB   sav;
      L     2.000000e+000;
      /R    ;
sav:  T     #tmpHys;

NETWORK
TITLE =

      L     #rSOLL; // Sollwert
      L     #tmpHys; // Hystersewert
      +R    ;
      T     #rMax; // Ausgang max. Wert
      POP   ; // Sollwert zurück in AKKU1
      L     #rSOLL; // Sollwert
      L     #tmpHys; // Hystersewert
      -R    ;
      T     #rMin; // Ausgang min. Wert
END_FUNCTION

FUNCTION "m7b_GetParity_DWORD" : BOOL
TITLE =Get ParityBit for Even/Odd Parity and count Hi-Bits (0..32)
//AUTOR: Stefan Maag, Dipl.-Ing. (FH) Elektrotechnik
//DATUM: 4/2020
//
//RET_VAL : Parity Bit, so dass gewünschte gerade/ungerade Parität entsteht
//FC_ENO  : TRUE: mindestens 1 Bit war Hi
//
//Für BYTE/INT/DINT/REAL, diese zuerst auf ein DWORD kopieren bzw. wandeln
//
//AENDERUNGSVERMERKE:
//--------------------------------------------------------------------------------
//DATUM       NAME       AENDERUNG
//--------------------------------------------------------------------------------
//03.04.2020  S.Maag     Entsand aus BitCountINT
//--------------------------------------------------------------------------------
//
//HINWEISE:
AUTHOR : 'S.Maag'
FAMILY : Maagic7
VERSION : 0.1


VAR_INPUT
  dwVAL : DWORD ;	//zu prüfender Wert
  cfg_Even_Odd : BOOL ;	//FALSE: returns odd parity; TRUE: returns even parity
END_VAR
VAR_OUTPUT
  iBitCount : INT ;	//No of Hi-Bits
END_VAR
VAR_TEMP
  AR1 : DWORD ;
  EvenParity : BOOL ;
END_VAR
BEGIN
NETWORK
TITLE =Anzahl der gestzten Bits in INT Zählen
//Die Anzahl der Bits wird dann in #Bits zurückgeben, steht aber auch noch
//zusätzlich im Akku1 zur Verfügung
      TAR1  #AR1; // Adressregister im TMEP-Bereich sichern
      L     #dwVAL; // zu prüfenden Wert in Akku 1
      L     DW#16#0; // Adressregister 1 wird als BitZaehler verwendet
      LAR1  ; // daher auf 0 setzten
LOOP: TAK   ; // zu prüfende Bits wieder in Akku 1
      SRD   1; // erstes zu Prüfendes Bit hinausschieben
      SPZ   NEXT; // Wenn 0 dann Schleifenende prüfen
      +AR1  P#0.1; // Bitzähler im Adressregister 1 um 1 erhöhen
NEXT: L     DW#16#0; // Vergleichswert, Bits zählen bis 0 erreicht
      <>D   ; // Solange wiederholen bis zu prüfende Bits
      SPB   LOOP; // den Wert 0 erreicht haben, alle Bits gezählt!
      TAR1  ; // Anzahl Bits aus Adressregister in Akku 1
      <>D   ; // Anzahl Bits auf 0 prüfen (mit vorheriger 0, bereits im AKKU)
      SAVE  ; // BIE-BIT = High, wenn Anzahl der Bits<>0
      CLR   ; // VKE wieder rücksetzen (verarbeiten)
      T     #iBitCount; // Anzahl Bits in Rückgabewert
      SRD   1; // erstes Bit der Bitanzahl rausschieben
      U     ==0; // Wenn Bit=0, dann gerade Bitanzahl
      =     #EvenParity;
// Parity Bit für gewünsche Parity erzeugen
      UN    #EvenParity; // Parity ist nicht gerade (ungerade)
      UN    #cfg_Even_Odd; // und gerade Parity gefordert
      O     ;
      U     #EvenParity; // Parity ist gerade
      U     #cfg_Even_Odd; // ungerade Parity ist gefordert
      =     #RET_VAL; // Parity Bit, so dass geforderte Parity erziehlt wird

      LAR1  #AR1; // Adressregister wieder herstellen

NETWORK
TITLE =alternativer Code
//    // #BitCounter & #LoopRegister im TEMP-Bereich als INT anlegen
//
//      L     0
//      T     #BitCounter                 // Anzahl Bits auf 0
//      L     2#1000000000000000          // SchleifenRegister
//      T     #LoopRegister               // initialisieren
//
//      L     #Wert                       // zu prüfenden Wert in Akku 1
//loop: SRD   1                           // 1 Bit hinausschieben
//      SPP   inc                         // wenn positiv, dann Bit zaehlen
//      SPA   next                        // sonst weiter mit Schleifenregister
//
//inc:  L     #BitCounter                 // Bit zählen
//      +     1
//      T     #BitCounter
//      TAK                               // zu prüfenden Wert in Akku 1 zurück
//
//next: L     #LoopRegister               // SchleifenRegister auf nächstes Bit
//      SRD   1
//      SPP   end                         // falls positiv, dann letztes Bit !=
//Ende
//      T     #LoopRegister
//      TAK
//      SPA   loop
//
//end:  L     #BitCounter                 // Anzahl Bits zurückgeben
//      T     #Bits
//      L     0                           // BIE-Bit=High, wenn Anzahl Bits >0
//      <>I
//      SAVE
//      CLR
//


END_FUNCTION

FUNCTION "m7b_GetFirstOf8Bits" : VOID
TITLE =Get First Hi of 8 Bits
//AUTOR: Stefan Maag, Dipl.-Ing. (FH) Elektrotechnik
//DATUM: 6/2007
//INTERNET: www.maagic7.de
//
//AENDERUNGSVERMERKE:
//--------------------------------------------------------------------------------
//DATUM        NAME        AENDERUNG
//--------------------------------------------------------------------------------
//12.08.2013   S.Maag    direkets Byteweises kopieren von den Eingängen
//                       funktioniert nur, wenn die Quellbits aufeinanderfolgend
//                       sind. (war bisher immer zufällig so, da KOP und
//                       Übergabe per Lx.y, Im AWL funktioniert es nicht, da
//                       direkte Merkeradressen übergeben werden)
//                       Bits müssen deshalb immer einzeln kopiert werden!
//--------------------------------------------------------------------------------
//
//HINWEISE:
AUTHOR : 'S.Maag'
FAMILY : Maagic7
VERSION : 0.1


VAR_INPUT
  RESET : BOOL ;
  Sig1 : BOOL ;
  Sig2 : BOOL ;
  Sig3 : BOOL ;
  Sig4 : BOOL ;
  Sig5 : BOOL ;
  Sig6 : BOOL ;
  Sig7 : BOOL ;
  Sig8 : BOOL ;
END_VAR
VAR_OUTPUT
  TheByte : BYTE ;	//The 8 Input Bits as Byte
  iNoOf1st : INT ;	//No of 1st Hi-Signal 1..8 (0 = no Hi Bit)
END_VAR
BEGIN
NETWORK
TITLE =

      UN    #RESET;
      SPB   ne1;

      L     0;
      T     #TheByte;
      T     #iNoOf1st;

      CLR   ;
      SAVE  ;
      BEA   ;
ne1:  NOP   0;

NETWORK
TITLE =
//
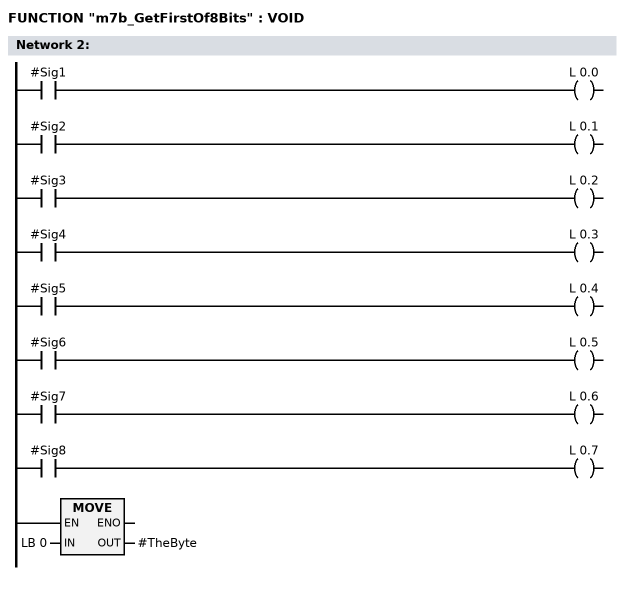
      U     #Sig1;
      =     L      0.0;
      U     #Sig2;
      =     L      0.1;
      U     #Sig3;
      =     L      0.2;
      U     #Sig4;
      =     L      0.3;
      U     #Sig5;
      =     L      0.4;
      U     #Sig6;
      =     L      0.5;
      U     #Sig7;
      =     L      0.6;
      U     #Sig8;
      =     L      0.7;

      L     LB     0;
      T     #TheByte;

NETWORK
TITLE =Nr des ersten gesetzten Bits
//CODE FROM FC192 m7a_FirstBit_INT
      L     LB     0; // zu prüfenden Wert in Akku
      L     0; // vergleichen ob Wert = 0
      <>I   ; // dann Ende, wenn nicht muss mind. 1 Bit gesetzt sein
      SAVE  ; // Anzahl Bits <> 0 in BIE-Bit speichern
      SPBN  end; // ENDE, wenn Wert = 0
      INC   1; // Schleifenzaehler in Akku 1 auf 1 stellen = BitPosition
      TAK   ; // zu prüfende Bits in Akku 1 zurück
Loop: SRW   1; // 1 Bit hinausschieben
      SPP   save; // wenn poitiv, dann erstes Bit gefunden => speichern
      TAK   ; // Schleifenzaehler in Akku 1
      INC   1; // erhöhen Schleifenzaehler, BitNr.
      TAK   ; // zu prüfende Bits in Akku zurück
      SPA   Loop; // Schleife für nächstes Bit wiederholen
save: TAK   ; // Schleifenzaehler, BitNr in Akku 1
end:  T     #iNoOf1st; // BitPosition zurückgeben


NETWORK
TITLE =

      SET   ;
      SAVE  ;
      CLR   ;


END_FUNCTION

FUNCTION "m7b_FSM_STATE_TIME" : VOID
TITLE =Count Time pulses of State No.
//Erfasst die Zeit der Schrittkette im akutellen Schritt.
//Zeitbasis muss als Taktflankenmerker übergeben werden.
//So lassen sich z.B. 0.1sec und 1sec Taktungen erreichen, je nachdem welchen
//Basistakt man wählt.
//
//ENO: True for 1 cycle, if StateNo change (=Timer Restart / RESET)
//
//AUTOR: Stefan Maag, Dipl.-Ing. (FH) Elektrotechnik
//DATUM: 2/2017
//
//AENDERUNGSVERMERKE:
//--------------------------------------------------------------------------------
//DATUM        NAME            AENDERUNG
//--------------------------------------------------------------------------------
//
//--------------------------------------------------------------------------------
//
//HINWEISE:
//
AUTHOR : 'S.Maag'
FAMILY : Maagic7
VERSION : 0.1


VAR_INPUT
  TaktImpuls : BOOL ;	//Taktimpuls 1sec
  iSNR : INT ;	//Schrittnummer / State No.
END_VAR
VAR_OUTPUT
  dTime_10xTakt : DINT ;	//Zähler Zeitimpulse (10xTakt, sec) / Counter Time pulses (10xTakt, sec)
END_VAR
VAR_IN_OUT
  io_dTime_TAKT : DINT ;	//Zähler Zeitimpulse (Takt, 1/10sec) / Counter Time pulses (takt 1/10sec)
  io_iMemSNR : INT ;	//Speicher letzte Schrittnummer / Memory last State No.
END_VAR
VAR_TEMP
  tmpMSG_RESET : BOOL ;
END_VAR
BEGIN
NETWORK
TITLE =



NETWORK
TITLE =Reset Time when State No changed
//Achtung: direkts (SAVE) hier statt tmpMSG_RESET
//geht nicht. Sonst werden nachfolgende Verknüpfungen mit
//nicht ausgeführt, das das BIE-Bit automatisch mit verknüpft wird.
//Es wäre vorher ein CLR nötig
      U(    ;
      U(    ;
      L     #iSNR;
      L     #io_iMemSNR;
      <>I   ;
      )     ;
      SPBNB _001;
      L     L#0;
      T     #io_dTime_TAKT;
      SET   ;
      SAVE  ;
      CLR   ;
_001: U     BIE;
      )     ;
      SPBNB _002;
      L     #iSNR;
      T     #io_iMemSNR;
      SET   ;
      SAVE  ;
      CLR   ;
_002: U     BIE;
      =     #tmpMSG_RESET;
NETWORK
TITLE =Count Time

      U     #TaktImpuls;
      SPBNB _003;
      L     #io_dTime_TAKT;
      L     L#1;
      +D    ;
      T     #io_dTime_TAKT;
_003: NOP   0;
NETWORK
TITLE =Time 10xTakt

      L     #io_dTime_TAKT;
      L     L#10;
      /D    ;
      T     #dTime_10xTakt;
      NOP   0;
NETWORK
TITLE =RESET / RESTART Message as FC-ENO

      U     #tmpMSG_RESET;
      SAVE  ;
END_FUNCTION

FUNCTION "m7b_FSM_TIME" : VOID
TITLE =Count Time pulses of active State range
//Duration of active States
//starts at: StateNo = iStateStart
//stops at:  StateNo = iStateEnd
//
//Ermittelt die abgelaufene Zeit einer Schrittkette von
//iStateStart bis iStateEnd. Anwendung z.B. zur Laufzeitüberwachung!
//
//AUTOR: Stefan Maag, Dipl.-Ing. (FH) Elektrotechnik
//DATUM: 11/2017
//
//AENDERUNGSVERMERKE:
//--------------------------------------------------------------------------------
//DATUM        NAME            AENDERUNG
//--------------------------------------------------------------------------------
//
//--------------------------------------------------------------------------------
//
//HINWEISE:
AUTHOR : 'S.Maag'
FAMILY : Maagic7
VERSION : 0.1


VAR_INPUT
  TaktImpuls : BOOL ;	//Taktimpuls 1sec
  iSNR : INT ;	//Schrittnummer / State No.
  iStateStart : INT ;
  iStateEnd : INT ;
END_VAR
VAR_OUTPUT
  dTime_10xTakt : DINT ;	//Zähler Zeitimpulse (10xTakt, sec) / Counter Time pulses (10xTakt, sec)
END_VAR
VAR_IN_OUT
  io_dTime_TAKT : DINT ;	//Zähler Zeitimpulse (Takt, 1/10sec) / Counter Time pulses (takt 1/10sec)
  io_iMemSNR : INT ;	//Speicher letzte Schrittnummer / Memory last State No.
END_VAR
VAR_TEMP
  MSG_active : BOOL ;
END_VAR
BEGIN
NETWORK
TITLE =



NETWORK
TITLE =State No in the active range => cout Time
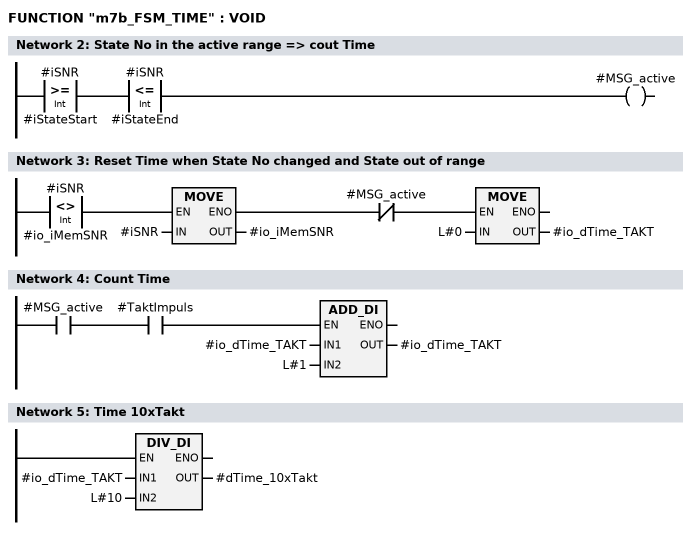

      U(    ;
      L     #iSNR;
      L     #iStateStart;
      >=I   ;
      )     ;
      U(    ;
      L     #iSNR;
      L     #iStateEnd;
      <=I   ;
      )     ;
      =     #MSG_active;
NETWORK
TITLE =Reset Time when State No changed and State out of range

      U(    ;
      U(    ;
      L     #iSNR;
      L     #io_iMemSNR;
      <>I   ;
      )     ;
      SPBNB _001;
      L     #iSNR;
      T     #io_iMemSNR;
      SET   ;
      SAVE  ;
      CLR   ;
_001: U     BIE;
      )     ;
      UN    #MSG_active;
      SPBNB _002;
      L     L#0;
      T     #io_dTime_TAKT;
_002: NOP   0;
NETWORK
TITLE =Count Time

      U     #MSG_active;
      U     #TaktImpuls;
      SPBNB _003;
      L     #io_dTime_TAKT;
      L     L#1;
      +D    ;
      T     #io_dTime_TAKT;
_003: NOP   0;
NETWORK
TITLE =Time 10xTakt

      L     #io_dTime_TAKT;
      L     L#10;
      /D    ;
      T     #dTime_10xTakt;
      NOP   0;
NETWORK
TITLE =FC-ENO


      U     #MSG_active;
      SAVE  ;
END_FUNCTION

FUNCTION "m7b_GlobalParent_Mode" : VOID
TITLE =Get Global/Parent Control Mode
//Get the Global or Parent Control mode to set the device mode
//
//[IN]
//iGlobalMode: The Global Control Mode which sets the User Rights for operation
//             0: all operation allowed (OFF/ON/AUTO)
//             1: only HAND (OFF/ON) allowed, AUTO is disabled
//             2: Global Control AUTO; no user Operation allowed, set fix to AUTO
//
//iParentMode: The actual Mode of the Parent Control
//             The Child Device is controled with the Mode of the Parent Device
//             0: OFF (HAND_OFF)
//             1: ON  (HAND_ON)
//             2: AUTO
//
//cfg_Global_Parent: Select the Device Control Mode
//     FALSE : The Device is controled according to the Globel User Right's
//             iGlobalMode is used to set the DeviceMode
//
//     TRUE :  The Device is controled directly/simultaneously with the mode of a
//             Parent Control. The Actual Device is a Child Device
//             iParentMode is used to set the DeviceMode
//
//ioHMIactivate: HMI Button OFF/ON/AUTO: 0=hide; 1=visible
//               In HMI, a click on the device (valve, motor ...) must toggle
//               this switch between 0 and 1.
//               Then the output HMI_ButtonStyle change between visible and
//               unvisible.
//               This function helps to not confuse the user with tons of
//               visible buttons.
//               If manual operation is enabled, the user must click on the device
//               to show the manual operation button for the device.
//
//AUTOR: Stefan Maag, Dipl.-Ing. (FH) Elektrotechnik
//DATUM: 9/2018
//
//AENDERUNGSVERMERKE:
//--------------------------------------------------------------------------------
//DATUM        NAME        AENDERUNG
//--------------------------------------------------------------------------------
//20.11.2019   S.Maag    Seperate HMI_Button "ioHMIactive" to activate and
//                       deactivate the OFF_ON_AUTO Button.
//                       In HMI, a click on the device (valve, motor ...) must
//                       toggle this switch between 0 and 1.
//
//                       Outuput "HMI_Button_Style" to control OFF_ON_AUTO
//                       Button style.
//--------------------------------------------------------------------------------
//
//HINWEISE:
//             Use this mode, if you want to control maybe a valve
//             simultan with a Pump.
//
AUTHOR : 'S.Maag'
FAMILY : Maagic7
VERSION : 0.1


VAR_INPUT
  iGlobalMode : INT ;	//0: Allow all / 1: Global HAND (AUTO forbidden) / 2: Global AUTO
  iParentMode : INT ;	//Mode of the Parent Control
  cfg_Global_Parent : BOOL ;	//0: Device controled by Global Control; 1:=Device conrolled by Parent Device
END_VAR
VAR_OUTPUT
  SET_OFF : BOOL ;
  SET_HAND : BOOL ;
  SET_AUTO : BOOL ;	//Set Device Mode fix to AUTO (User operation HAND OFF/ON not allowed)
  ENABLE_AUTO : BOOL ;	//Enable the AUTO MODE selection for the User
  HMI_ButtonStyle : INT ;	//Value to display HMI Button (0: All; 1: OFF/ON; 2: Hide)
END_VAR
VAR_IN_OUT
  ioHMIactivate : INT ;	//HMI Button OFF/ON/AUTO: 0=hide; 1=visible
END_VAR
BEGIN
NETWORK
TITLE =
//0 : Allow all User Operation
//1 : Global Hand Mode (dont allow Auto Operation)
//2 : Global Auto Mode


NETWORK
TITLE =ENABLE AUTO
//in Mode 0 user can operate all (OFF/ON/AUTO)
//in Mode 2 user can't operate anything (Set the device fix to AUTO)
//          so Auto must be ENABLED
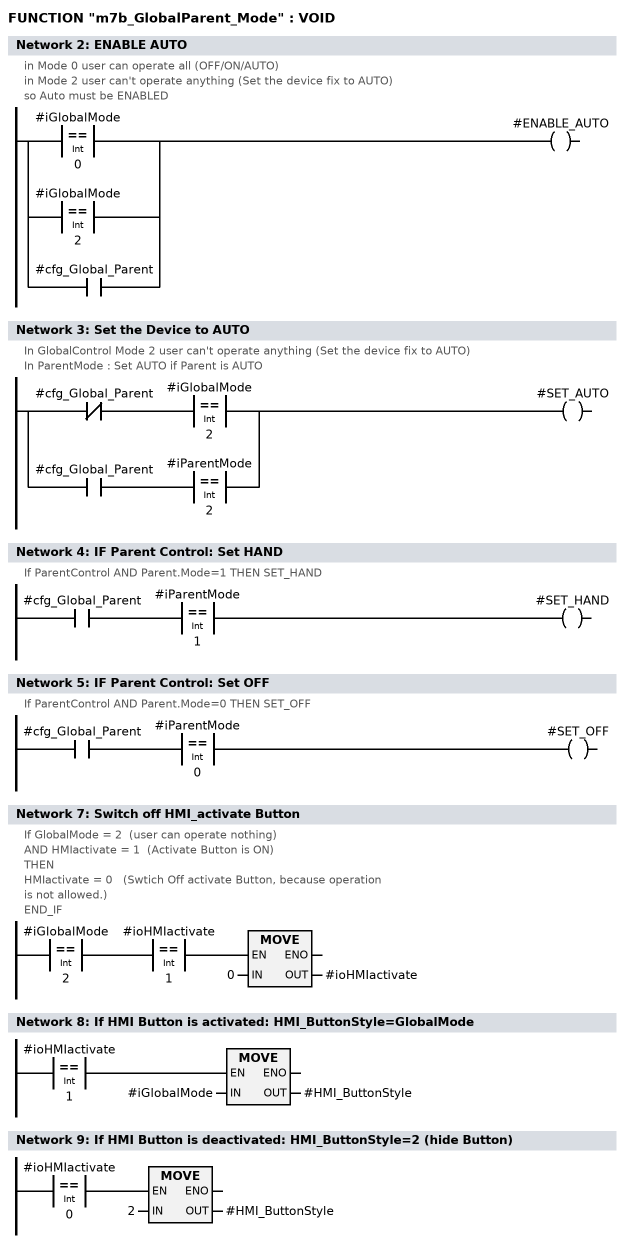


      O(    ;
      L     #iGlobalMode;
      L     0;
      ==I   ;
      )     ;
      O(    ;
      L     #iGlobalMode;
      L     2;
      ==I   ;
      )     ;
      O     #cfg_Global_Parent;
      =     #ENABLE_AUTO;
NETWORK
TITLE =Set the Device to AUTO
//In GlobalControl Mode 2 user can't operate anything (Set the device fix to AUTO)
//In ParentMode : Set AUTO if Parent is AUTO
      UN    #cfg_Global_Parent;
      U(    ;
      L     #iGlobalMode;
      L     2;
      ==I   ;
      )     ;
      O     ;
      U     #cfg_Global_Parent;
      U(    ;
      L     #iParentMode;
      L     2;
      ==I   ;
      )     ;
      =     #SET_AUTO;
NETWORK
TITLE =IF Parent Control: Set HAND
//If ParentControl AND Parent.Mode=1 THEN SET_HAND
      U     #cfg_Global_Parent;
      U(    ;
      L     #iParentMode;
      L     1;
      ==I   ;
      )     ;
      =     #SET_HAND;
NETWORK
TITLE =IF Parent Control: Set OFF
//If ParentControl AND Parent.Mode=0 THEN SET_OFF
      U     #cfg_Global_Parent;
      U(    ;
      L     #iParentMode;
      L     0;
      ==I   ;
      )     ;
      =     #SET_OFF;
NETWORK
TITLE =HMI activate Button
//======================================================================
//                    HMI activate Button
//======================================================================
//
//with click on the device (valve, motor) the HMI activate button is
//switched on/off. With activated signal, the button for OFF/ON/AUTO
//is visible.
NETWORK
TITLE =Switch off HMI_activate Button
//If GlobalMode = 2  (user can operate nothing)
//   AND HMIactivate = 1  (Activate Button is ON)
//
//THEN
//   HMIactivate = 0   (Swtich Off activate Button, because operation
//                      is not allowed.)
//
//END_IF
      U(    ;
      L     #iGlobalMode;
      L     2;
      ==I   ;
      )     ;
      U(    ;
      L     #ioHMIactivate;
      L     1;
      ==I   ;
      )     ;
      SPBNB _001;
      L     0;
      T     #ioHMIactivate;
_001: NOP   0;
NETWORK
TITLE =If HMI Button is activated: HMI_ButtonStyle=GlobalMode

      U(    ;
      L     #ioHMIactivate;
      L     1;
      ==I   ;
      )     ;
      SPBNB _002;
      L     #iGlobalMode;
      T     #HMI_ButtonStyle;
_002: NOP   0;
NETWORK
TITLE =If HMI Button is deactivated: HMI_ButtonStyle=2 (hide Button)

      U(    ;
      L     #ioHMIactivate;
      L     0;
      ==I   ;
      )     ;
      SPBNB _003;
      L     2;
      T     #HMI_ButtonStyle;
_003: NOP   0;
END_FUNCTION

FUNCTION "m7b_RP_FILL_INT" : VOID
TITLE =Ringpuffer mit Wert fuellen
//AUTOR: Stefan Maag, Dipl.-Ing. (FH) Elektrotechnik
//DATUM: 8/2017
//INTERNET: www.maagic7.de
//
//AENDERUNGSVERMERKE:
//--------------------------------------------------------------------------------
//DATUM        NAME        AENDERUNG
//--------------------------------------------------------------------------------
//
//--------------------------------------------------------------------------------
//
//HINWEISE:
AUTHOR : 'S.Maag'
FAMILY : Maagic7
VERSION : 0.1


VAR_INPUT
  DB_RP : BLOCK_DB ;
  iFillVavlue : INT ;	//Fuellwert
  idxSTART : INT ;	//Start bei Index (0..255)
  iAnzahl : INT ;	//Anzahl zu schreibender Werte (0..256)
  cfg_REV_FWD : BOOL ;	//Konfiguration Richtung: 0: Füllen rückwärts; 1: füllen vorwärts
END_VAR
VAR_TEMP
  tmpLOP : INT ;
  tmpPtr : INT ;
END_VAR
BEGIN
NETWORK
TITLE =

      CLR   ;
      SAVE  ;

NETWORK
TITLE =

      AUF   #DB_RP; // Ringpuffer DB öffnen

      L     #idxSTART;
      T     #tmpPtr;


      L     #iAnzahl;
      L     0;
      <=I   ;
      SPB   END; // Wenn Anzahl <=0, dann nichts tun => ENDE

      L     #iAnzahl;
      L     256;
      >I    ;
      SPB   LOOP; // Wenn >256, dann auf 256 begrenzen
      TAK   ;
LOOP: T     #tmpLOP; // Schleifenzaehler
      L     #tmpPtr; // Indexwert Ringpuffer 0..255
      PUSH  ; // copy tmpPtr to AKKU2
      U     #cfg_REV_FWD; // Wenn fuellen vorwaerts
      SPB   fwd;
      DEC   1; // tmpPtr-- (255..0); fuellen rueckwaerts
      SPA   save;
fwd:  INC   1; // tmpPtr++ (0..255); fuellen vorwaerts
save: T     #tmpPtr;
      TAK   ; // org tmpPtr => AKKU 1
      SLD   4; // SLD 1 wegen INT-Werten=>Byte + SLD 3 wegen Pointer
      L     P#0.0; // 0-Pointer addieren
      +D    ; // Pointer auf Daten erzeugen
      LAR1  ; // in Adressregister 1 laden

      L     #iFillVavlue; // Eingangswert laden
      T     DBW [AR1,P#0.0]; // in DB speichern

      L     #tmpLOP; // Schleifenzaehler
      LOOP  LOOP; // LOOP:= AKKU 1, springe wenn <>0

      SET   ;
      SAVE  ;
      CLR   ;
END:  NOP   0;
END_FUNCTION

FUNCTION "m7b_POSITONIEREN_REAL" : VOID
TITLE =Positionierrichtung Achse ermitteln. Position ok ausgeben
//Dieser FC ermittelt die Positonierrichtung von Achsen (vorw./rückw.)
//
//TOL_POS : Ist die zuslässige Positionsdifferenz, ab der die Achse zum
//          nachpositionieren anfängt
//
//TOL_POS_OK : Ist die zulässige Toleranz bis zu der gemeldet wird, dass
//             die Achse im gültigen Positiosfenster steht
//
//AUTOR: Stefan Maag, Dipl.-Ing. (FH) Elektrotechnik
//DATUM: 12/2012
//INTERNET: www.maagic7.de
//
//AENDERUNGSVERMERKE:
//--------------------------------------------------------------------------------
//DATUM        NAME        AENDERUNG
//--------------------------------------------------------------------------------
//
//--------------------------------------------------------------------------------
//
//HINWEISE:
//Funktion identisch FC96 Positionierrichtung DINT
AUTHOR : 'S.Maag'
FAMILY : Maagic7
VERSION : 0.1


VAR_INPUT
  FRG : BOOL ;	//Freigabe
  SOLL : REAL ;	//Sollwert
  IST : REAL ;	//Istwert Achse
  TOL_POS_OK : REAL ;	//Toleranz für Position ok Meldung
  TOL_POS : REAL ;	//Toleranz Posiitionierung Achse
END_VAR
VAR_OUTPUT
  PLUS : BOOL ;
  MINUS : BOOL ;
  POS_OK : BOOL ;
END_VAR
BEGIN
NETWORK
TITLE =Postion Achse prüfen, Positionsdifferenz

      L     #SOLL; // aktuelle Sollposition
      L     #IST; // aktuelle Istposition
      -R    ; // Positionierdifferenz
      SPP   PLUS;
      NEGR  ; // nach positiv

PLUS: L     #TOL_POS_OK; // Toleranz für Position ok
      <R    ;
      =     #POS_OK; // Ausgang Position ok

      TAK   ; // Positionsdifferenz in AKKU1
      L     #TOL_POS; // Toleranz für Positionierung
      <R    ;
      SAVE  ;
      SPB   STOP; // Innerhalb Toleranz, dann Stop

NETWORK
TITLE =FREIGABE

      UN    #FRG; // keine Freigabe, dann Stop
      SPB   STOP;

NETWORK
TITLE =Postionierrichtung vorw. oder rückw.

      L     #SOLL; // Soll
      L     #IST; // IST
      >R    ;
      SPB   VW; // Soll > Ist, dann vw
      SPA   RW; // sonst rw
NETWORK
TITLE =Richtungsausgänge setzen

STOP: R     #PLUS;
      R     #MINUS;
      BEA   ;

VW:   R     #MINUS;
      S     #PLUS;
      BEA   ;

RW:   R     #PLUS;
      S     #MINUS;
      BE    ;
END_FUNCTION

FUNCTION_BLOCK "m7b_6x_MSG_QUITT"
TITLE =6 Meldungen mit Quittierung
//6 Meldungen speichernd verarbeiten.
//
//cfg_HIDE: ist der Konfigurationseingang cfg_HIDE Hi, dann werden Meldungen
//          Folgemeldungen ausgeblendet. D.h. Meldung die weiter oben steht
//          sperrt nachfolgende.
//
//Quittierung mit RESET (für Autoquittierung RESET:=TRUE)
//
//Verwendung:
//Motoren mit mehreren Störmeldungen (Motorschutzschalter, Endschalter)
//(Pumpen mit Trockenlaufschutz, Drucküberwachung)
//
//FB-ENO: TRUE
//
//AUTOR: Stefan Maag, Dipl.-Ing. (FH) Elektrotechnik
//DATUM: 10/2012
//
//AENDERUNGSVERMERKE:
//--------------------------------------------------------------------------------
//DATUM        NAME            AENDERUNG
//--------------------------------------------------------------------------------
//16.03.2020   S.Maag     FC.ENO = UN IN_MSG0 .. IN MSG5 (kein Meldeeingang aktiv)
//                        dies kann verwendet werden, um AutoReset nach Zeit
//                        durchzuführen, wenn alle Fehlermeldungen aus!
//
//03.09.2018   S.Maag     FC.ENO = TRUE; (war FC.ENO=MSG_OK)
//
//17.10.2014   S.Maag     Ab MSG_3 das F für Folgemeldung entfernt, da schon
//                        seit beginn alle Meldungen als Folgemeldung abgeschaltet
//                        werden können.
//--------------------------------------------------------------------------------
//
//HINWEISE:
AUTHOR : 'S.Maag'
FAMILY : Maagic7
VERSION : 0.1


VAR_INPUT
  IN_MSG_0 : BOOL ;	//Signal Meldung 0:
  IN_MSG_1 : BOOL ;	//Signal Meldung 1:
  IN_MSG_2 : BOOL ;	//Signal Meldung 2:
  IN_MSG_3 : BOOL ;	//Signal Meldung 3:
  IN_MSG_4 : BOOL ;	//Signal Meldung 4:
  IN_MSG_5 : BOOL ;	//Signal Meldung 5:
  RESET : BOOL ;	//RESET: für Autoquittierung fest auf Hi
  cfg_HIDE : BOOL ;	//Konfigurationseingang Folgemeldungen ausblenden
END_VAR
VAR_OUTPUT
  OUT_MSG_0 : BOOL ;	//Ausgang Meldung 0
  OUT_MSG_1 : BOOL ;	//Ausgang Meldung 1
  OUT_MSG_2 : BOOL ;	//Ausgang Meldung 2
  OUT_MSG_3 : BOOL ;	//Ausgang Meldung 3
  OUT_MSG_4 : BOOL ;	//Ausgang Meldung 4
  OUT_MSG_5 : BOOL ;	//Ausgang Meldung 5
  OUT_MSG : BOOL ;	//Sammelmeldung: True, wenn Meldung vorhanden
  OUT_OK : BOOL ;	//Keine Meldung: True, wenn keine Meldung aktiv
  FLAGS : BYTE ;	//Meldebits gesammelt in Byte
END_VAR
VAR_TEMP
  HM_MSG_ON : BOOL ;
END_VAR
BEGIN
NETWORK
TITLE =



NETWORK
TITLE =Meldung 0
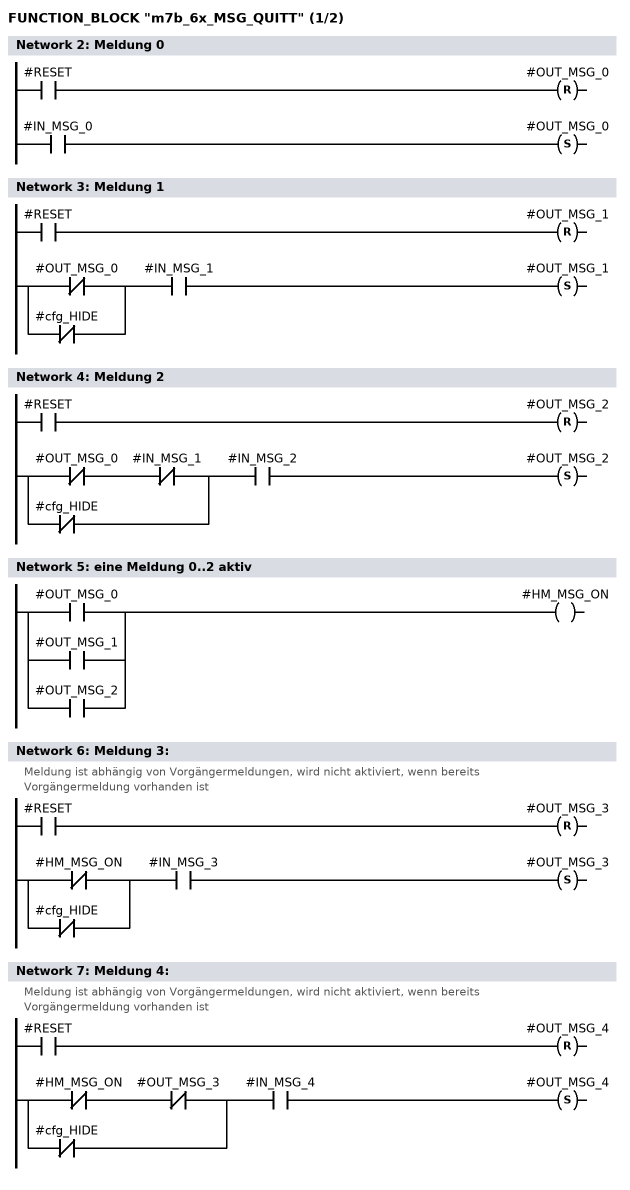

      U     #RESET;
      R     #OUT_MSG_0;
      U     #IN_MSG_0;
      S     #OUT_MSG_0;
      NOP   0;
NETWORK
TITLE =Meldung 1

      U     #RESET;
      R     #OUT_MSG_1;
      U(    ;
      ON    #OUT_MSG_0;
      ON    #cfg_HIDE;
      )     ;
      U     #IN_MSG_1;
      S     #OUT_MSG_1;
      NOP   0;
NETWORK
TITLE =Meldung 2

      U     #RESET;
      R     #OUT_MSG_2;
      U(    ;
      UN    #OUT_MSG_0;
      UN    #IN_MSG_1;
      ON    #cfg_HIDE;
      )     ;
      U     #IN_MSG_2;
      S     #OUT_MSG_2;
      NOP   0;
NETWORK
TITLE =eine Meldung 0..2 aktiv

      O     #OUT_MSG_0;
      O     #OUT_MSG_1;
      O     #OUT_MSG_2;
      =     #HM_MSG_ON;
NETWORK
TITLE =Meldung 3:
//Meldung ist abhängig von Vorgängermeldungen, wird nicht aktiviert, wenn bereits
//Vorgängermeldung vorhanden ist
      U     #RESET;
      R     #OUT_MSG_3;
      U(    ;
      ON    #HM_MSG_ON;
      ON    #cfg_HIDE;
      )     ;
      U     #IN_MSG_3;
      S     #OUT_MSG_3;
      NOP   0;
NETWORK
TITLE =Meldung 4:
//Meldung ist abhängig von Vorgängermeldungen, wird nicht aktiviert, wenn bereits
//Vorgängermeldung vorhanden ist
      U     #RESET;
      R     #OUT_MSG_4;
      U(    ;
      UN    #HM_MSG_ON;
      UN    #OUT_MSG_3;
      ON    #cfg_HIDE;
      )     ;
      U     #IN_MSG_4;
      S     #OUT_MSG_4;
      NOP   0;
NETWORK
TITLE =Meldung 5:
//Meldung ist abhängig von Vorgängermeldungen, wird nicht aktiviert, wenn bereits
//Vorgängermeldung vorhanden ist
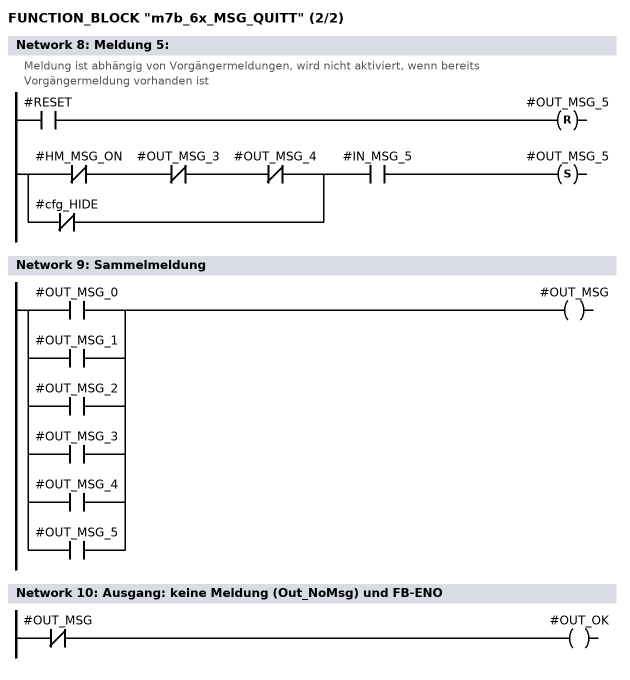
      U     #RESET;
      R     #OUT_MSG_5;
      U(    ;
      UN    #HM_MSG_ON;
      UN    #OUT_MSG_3;
      UN    #OUT_MSG_4;
      ON    #cfg_HIDE;
      )     ;
      U     #IN_MSG_5;
      S     #OUT_MSG_5;
      NOP   0;
NETWORK
TITLE =Sammelmeldung

      O     #OUT_MSG_0;
      O     #OUT_MSG_1;
      O     #OUT_MSG_2;
      O     #OUT_MSG_3;
      O     #OUT_MSG_4;
      O     #OUT_MSG_5;
      =     #OUT_MSG;
NETWORK
TITLE =Ausgang: keine Meldung (Out_NoMsg) und FB-ENO

      UN    #OUT_MSG;
      =     #OUT_OK;
NETWORK
TITLE =ENO = kein Meldeeingang aktiv
//16.03.2020 S.Maag
//
//Dies kann verwendet werden, um herauszufinden, wenn alle Meldeeingaenge wieder
//FALSE sind. Damit kann man dann z.B. einen AutoReset nach Zeit durchführen.
      UN    #IN_MSG_0;
      UN    #IN_MSG_1;
      UN    #IN_MSG_2;
      UN    #IN_MSG_3;
      UN    #IN_MSG_4;
      UN    #IN_MSG_5;
      SAVE  ;
NETWORK
TITLE =OUT MSG [0..7] als Byte nach Flags kopieren
//S.Maag 12.10.2012
//
//direktes laden über
//
//      L     P##OUT_MSG_0
//      LAR1
//      L     B [AR1,P#0.0]
//      T     #FLAGS
//
//funktioniert nich, da die Pointeradresse relativ zu den Instanzdaten ist
      L     B [AR2,P#2.0]; // in AR2 befindest sich immer der Pointer auf STAT Daten
      T     #FLAGS; // d.h. STAT Byte 2 laden und nach FLAGs


END_FUNCTION_BLOCK

FUNCTION_BLOCK "m7b_DelayedNiveau_REAL"
TITLE =Niveau-Schalter mit Min/Max Hysterese, Min- oder Max- schaltend
//Niveau-Schalter mit Delay, Min/Max Hysterese und Funktion Min- oder Max-
//schaltend
//
//VERWENDUNG:
//2-Punkt-Regler
//Befüllen oder entleeren von Tanks mit Füllstandsmesser
//Heizen bzw. kühlen
//
//VALUE : Istwert (Temperatur, Druck, Füllstand ...)
//MIN   : Minimalwert (Ein bei Min-schaltend bzw. Aus bei Max-schaltend)
//MAX   : Maximalwert (Aus bei Min-schaltend bzw. Ein bei Max-schaltend)
//
//Fkt_Min_Max:
//  0 = Minimumschaltend
//      Beim Minimum wird eingeschaltet bis das Maximum erreicht ist, dann aus
//      (z.B. befüllen, heizen)
//
//  1 = Maximumschaltend
//      Beim Maximu wird eingeschaltet bis das Minimum erreicht ist, dann aus
//      (z.B. entleeren, kühlen)
//
//OUT : Schaltsignal
//
//AUTOR: Stefan Maag, Dipl.-Ing. (FH) Elektrotechnik
//DATUM: 8/2013
//INTERNET: www.maagic7.de
//
//AENDERUNGSVERMERKE:
//--------------------------------------------------------------------------------
//DATUM        NAME        AENDERUNG
//--------------------------------------------------------------------------------
//28.08.2013   S.Maag      RESET-Eingang hinzugefügt
//--------------------------------------------------------------------------------
//
//HINWEISE: enstand aus FC84 'm7b_NiveauSchalter_REAL'
AUTHOR : 'S.Maag'
FAMILY : Maagic7
VERSION : 0.1


VAR_INPUT
  rVALUE : REAL ;	//Istwert
  rMIN : REAL ;	//Minimalwert Hysterese
  rMAX : REAL ;	//Maximalwert Hysterese
  cfg_Min_Max : BOOL ;	//0=MinSchaltend (z.B. befüllen, heizen) 1=MaxSchaltend (z.B. entleeren, kühlen)
  cfg_DELAY_OFF : BOOL ;	//TRUE: deaktiviert ON & OFF Verzögerung (für Programmgesteuerte Deaktivierung)
  RESET : BOOL ;	//RESET: löscht Ausgang
  timDelayOn : TIME ;	//Einschaltverzögerung: bei T=0 deaktiviert => unverz. schalten
  timDelayOff : TIME ;	//Ausschaltverzögerung: bei T=0 deaktiviert => unverz. schalten
END_VAR
VAR_OUTPUT
  OUT : BOOL ;	//Hilfsbit, Hilfmerker
  OnDelay : BOOL ;
  OffDelay : BOOL ;
  DSP_TIMER : TIME ;	//Anzeige Restlaufzeit bis schalten
END_VAR
VAR
  timDELAY : TIME ;
  TON_DELAY : "TON";
  Q_TON_DELAY : BOOL ;
  Q_DELAY : BOOL ;
  VAL_MIN : BOOL ;
  VAL_MAX : BOOL ;
END_VAR
VAR_TEMP
  ET_TIMER : TIME ;
END_VAR
BEGIN
NETWORK
TITLE =VALUE <= MIN
//Minimalwert erreicht:
//Einschaltpunkt bei Minimum schaltend
//Ausschaltpunkt bei Maximum schaltend
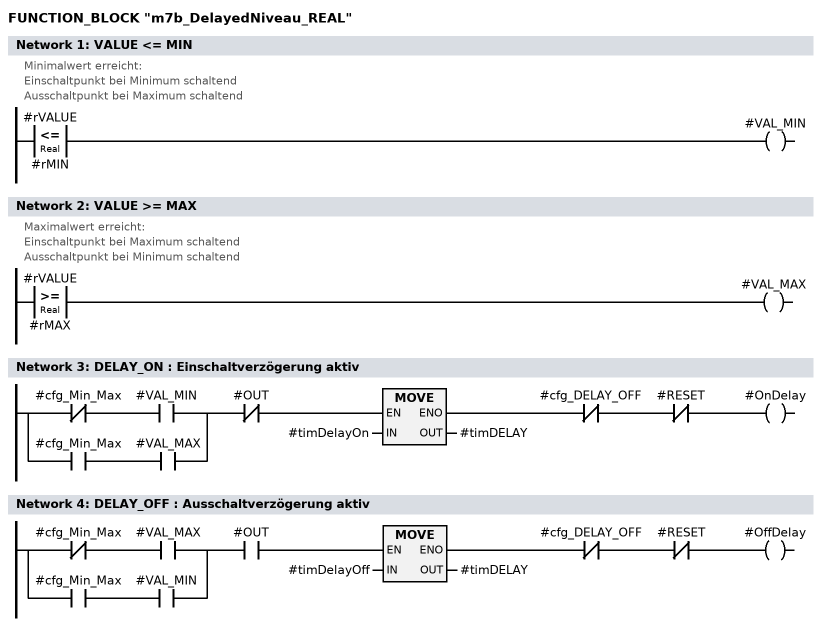
      L     #rVALUE;
      L     #rMIN;
      <=R   ;
      =     #VAL_MIN;
NETWORK
TITLE =VALUE >= MAX
//Maximalwert erreicht:
//Einschaltpunkt bei Maximum schaltend
//Ausschaltpunkt bei Minimum schaltend
      L     #rVALUE;
      L     #rMAX;
      >=R   ;
      =     #VAL_MAX;
NETWORK
TITLE =DELAY_ON : Einschaltverzögerung aktiv

      U(    ;
      U(    ;
      UN    #cfg_Min_Max;
      U     #VAL_MIN;
      O     ;
      U     #cfg_Min_Max;
      U     #VAL_MAX;
      )     ;
      UN    #OUT;
      SPBNB _001;
      L     #timDelayOn;
      T     #timDELAY;
      SET   ;
      SAVE  ;
      CLR   ;
_001: U     BIE;
      )     ;
      UN    #cfg_DELAY_OFF;
      UN    #RESET;
      =     #OnDelay;
NETWORK
TITLE =DELAY_OFF : Ausschaltverzögerung aktiv

      U(    ;
      U(    ;
      UN    #cfg_Min_Max;
      U     #VAL_MAX;
      O     ;
      U     #cfg_Min_Max;
      U     #VAL_MIN;
      )     ;
      U     #OUT;
      SPBNB _002;
      L     #timDelayOff;
      T     #timDELAY;
      SET   ;
      SAVE  ;
      CLR   ;
_002: U     BIE;
      )     ;
      UN    #cfg_DELAY_OFF;
      UN    #RESET;
      =     #OffDelay;
NETWORK
TITLE =Verzögerungszeit
//Falls DelayTime=0, muss Q_DELAY Hi werden.
//Da IEC-Timer bei T=0 einen RESET ausführen und Q=Lo ist, muss dieser Fall
//abgefangen werden.
//
      U(    ;
      U(    ;
      O     #OnDelay;
      O     #OffDelay;
      )     ;
      =     L      4.0;
      BLD   103;
      CALL #TON_DELAY (
           IN                       := L      4.0,
           PT                       := #timDELAY,
           Q                        := #Q_TON_DELAY,
           ET                       := #ET_TIMER);
      U     BIE;
      )     ;
      U(    ;
      O     #Q_TON_DELAY;
      O     #cfg_DELAY_OFF;
      O(    ;
      L     #timDELAY;
      L     0;
      ==D   ;
      )     ;
      )     ;
      =     #Q_DELAY;
NETWORK
TITLE =Anzeige Restlaufzeit TIMER
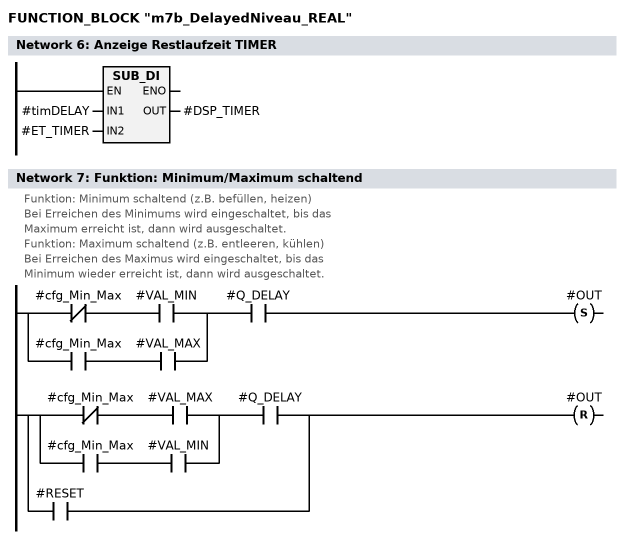

      L     #timDELAY;
      L     #ET_TIMER;
      -D    ;
      T     #DSP_TIMER;
      NOP   0;
NETWORK
TITLE =Funktion: Minimum/Maximum schaltend
//Funktion: Minimum schaltend (z.B. befüllen, heizen)
//Bei Erreichen des Minimums wird eingeschaltet, bis das
//Maximum erreicht ist, dann wird ausgeschaltet.
//
//Funktion: Maximum schaltend (z.B. entleeren, kühlen)
//Bei Erreichen des Maximus wird eingeschaltet, bis das
//Minimum wieder erreicht ist, dann wird ausgeschaltet.
      U(    ;
      UN    #cfg_Min_Max;
      U     #VAL_MIN;
      O     ;
      U     #cfg_Min_Max;
      U     #VAL_MAX;
      )     ;
      U     #Q_DELAY;
      S     #OUT;
      U(    ;
      U(    ;
      UN    #cfg_Min_Max;
      U     #VAL_MAX;
      O     ;
      U     #cfg_Min_Max;
      U     #VAL_MIN;
      )     ;
      U     #Q_DELAY;
      O     #RESET;
      )     ;
      R     #OUT;
      NOP   0;
NETWORK
TITLE =FB-ENO := TRUE

      SET   ;
      SAVE  ;
      CLR   ;

END_FUNCTION_BLOCK

FUNCTION_BLOCK "m7b_DelayedNiveau_INT"
TITLE =Niveau-Schalter mit Min/Max Hysterese, Min- oder Max- schaltend
//Niveau-Schalter mit Delay, Min/Max Hysterese und Funktion Min- oder Max-
//schaltend
//
//VERWENDUNG:
//2-Punkt-Regler
//Befüllen oder entleeren von Tanks mit Füllstandsmesser
//Heizen bzw. kühlen
//
//VALUE : Istwert (Temperatur, Druck, Füllstand ...)
//MIN   : Minimalwert (Ein bei Min-schaltend bzw. Aus bei Max-schaltend)
//MAX   : Maximalwert (Aus bei Min-schaltend bzw. Ein bei Max-schaltend)
//
//Fkt_Min_Max:
//  0 = Minimumschaltend
//      Beim Minimum wird eingeschaltet bis das Maximum erreicht ist, dann aus
//      (z.B. befüllen, heizen)
//
//  1 = Maximumschaltend
//      Beim Maximu wird eingeschaltet bis das Minimum erreicht ist, dann aus
//      (z.B. entleeren, kühlen)
//
//OUT : Schaltsignal
//
//AUTOR: Stefan Maag, Dipl.-Ing. (FH) Elektrotechnik
//DATUM: 8/2013
//INTERNET: www.maagic7.de
//
//AENDERUNGSVERMERKE:
//--------------------------------------------------------------------------------
//DATUM        NAME            AENDERUNG
//--------------------------------------------------------------------------------
//
//--------------------------------------------------------------------------------
//
//HINWEISE: enstand aus FC84 'm7b_NiveauSchalter_REAL'
AUTHOR : 'S.Maag'
FAMILY : Maagic7
VERSION : 0.1


VAR_INPUT
  iVALUE : INT ;	//Istwert
  iMIN : INT ;	//Minimalwert Hysterese
  iMAX : INT ;	//Maximalwert Hysterese
  cfg_Min_Max : BOOL ;	//0=MinSchaltend (z.B. befüllen, heizen) 1=MaxSchaltend (z.B. entleeren, kühlen)
  DELAY_OFF : BOOL ;	//TRUE: deaktiviert ON & OFF Verzögerung (für Programmgesteuerte Deaktivierung)
  timDelayOn : TIME ;	//Einschaltverzögerung: bei T=0 deaktiviert => unverz. schalten
  timDelayOff : TIME ;	//Ausschaltverzögerung: bei T=0 deaktiviert => unverz. schalten
END_VAR
VAR_OUTPUT
  OUT : BOOL ;	//Hilfsbit, Hilfmerker
  OnDelay : BOOL ;
  OffDelay : BOOL ;
  DSP_TIMER : TIME ;	//Anzeige Restlaufzeit bis schalten
END_VAR
VAR
  timDELAY : TIME ;
  TON_DELAY : "TON";
  Q_TON_DELAY : BOOL ;
  Q_DELAY : BOOL ;
  VAL_MIN : BOOL ;
  VAL_MAX : BOOL ;
END_VAR
VAR_TEMP
  ET_TIMER : TIME ;
END_VAR
BEGIN
NETWORK
TITLE =VALUE <= MIN
//Minimalwert erreicht:
//Einschaltpunkt bei Minimum schaltend
//Ausschaltpunkt bei Maximum schaltend
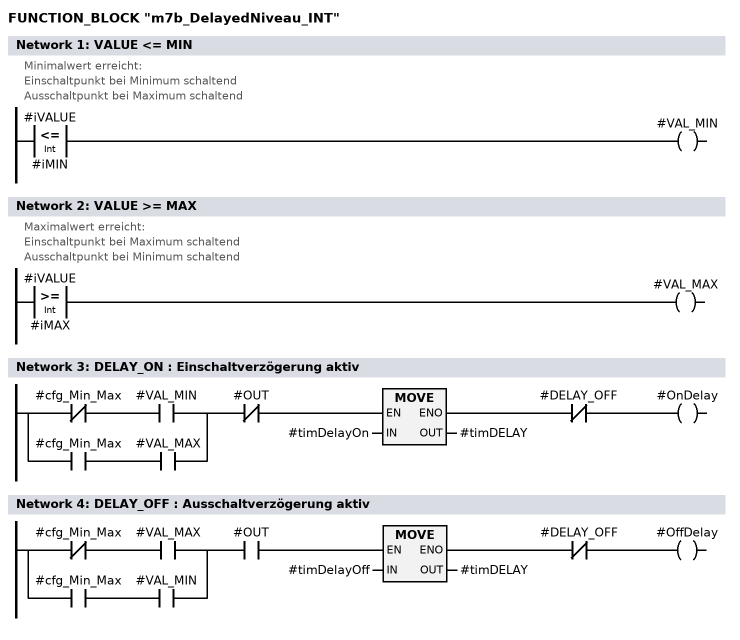
      L     #iVALUE;
      L     #iMIN;
      <=I   ;
      =     #VAL_MIN;
NETWORK
TITLE =VALUE >= MAX
//Maximalwert erreicht:
//Einschaltpunkt bei Maximum schaltend
//Ausschaltpunkt bei Minimum schaltend
      L     #iVALUE;
      L     #iMAX;
      >=I   ;
      =     #VAL_MAX;
NETWORK
TITLE =DELAY_ON : Einschaltverzögerung aktiv

      U(    ;
      U(    ;
      UN    #cfg_Min_Max;
      U     #VAL_MIN;
      O     ;
      U     #cfg_Min_Max;
      U     #VAL_MAX;
      )     ;
      UN    #OUT;
      SPBNB _001;
      L     #timDelayOn;
      T     #timDELAY;
      SET   ;
      SAVE  ;
      CLR   ;
_001: U     BIE;
      )     ;
      UN    #DELAY_OFF;
      =     #OnDelay;
NETWORK
TITLE =DELAY_OFF : Ausschaltverzögerung aktiv

      U(    ;
      U(    ;
      UN    #cfg_Min_Max;
      U     #VAL_MAX;
      O     ;
      U     #cfg_Min_Max;
      U     #VAL_MIN;
      )     ;
      U     #OUT;
      SPBNB _002;
      L     #timDelayOff;
      T     #timDELAY;
      SET   ;
      SAVE  ;
      CLR   ;
_002: U     BIE;
      )     ;
      UN    #DELAY_OFF;
      =     #OffDelay;
NETWORK
TITLE =Verzögerungszeit
//Falls DelayTime=0, muss Q_DELAY Hi werden.
//Da IEC-Timer bei T=0 einen RESET ausführen und Q=Lo ist, muss dieser Fall
//abgefangen werden.
//
      U(    ;
      U(    ;
      O     #OnDelay;
      O     #OffDelay;
      )     ;
      =     L      4.0;
      BLD   103;
      CALL #TON_DELAY (
           IN                       := L      4.0,
           PT                       := #timDELAY,
           Q                        := #Q_TON_DELAY,
           ET                       := #ET_TIMER);
      U     BIE;
      )     ;
      U(    ;
      O     #Q_TON_DELAY;
      O     #DELAY_OFF;
      O(    ;
      L     #timDELAY;
      L     0;
      ==D   ;
      )     ;
      )     ;
      =     #Q_DELAY;
NETWORK
TITLE =Anzeige Restlaufzeit TIMER
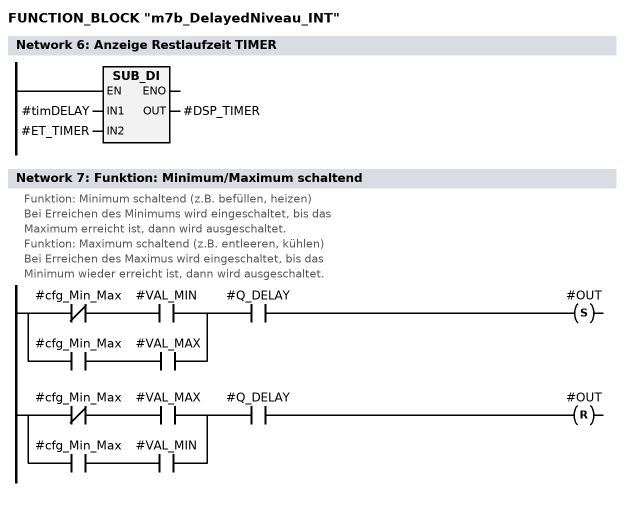

      L     #timDELAY;
      L     #ET_TIMER;
      -D    ;
      T     #DSP_TIMER;
      NOP   0;
NETWORK
TITLE =Funktion: Minimum/Maximum schaltend
//Funktion: Minimum schaltend (z.B. befüllen, heizen)
//Bei Erreichen des Minimums wird eingeschaltet, bis das
//Maximum erreicht ist, dann wird ausgeschaltet.
//
//Funktion: Maximum schaltend (z.B. entleeren, kühlen)
//Bei Erreichen des Maximus wird eingeschaltet, bis das
//Minimum wieder erreicht ist, dann wird ausgeschaltet.
      U(    ;
      UN    #cfg_Min_Max;
      U     #VAL_MIN;
      O     ;
      U     #cfg_Min_Max;
      U     #VAL_MAX;
      )     ;
      U     #Q_DELAY;
      S     #OUT;
      U(    ;
      UN    #cfg_Min_Max;
      U     #VAL_MAX;
      O     ;
      U     #cfg_Min_Max;
      U     #VAL_MIN;
      )     ;
      U     #Q_DELAY;
      R     #OUT;
      NOP   0;
NETWORK
TITLE =FB-ENO := TRUE

      SET   ;
      SAVE  ;
      CLR   ;

END_FUNCTION_BLOCK

FUNCTION_BLOCK "FIFO_INT_MIT_STARTW"
TITLE =FIFO mit Startwert, Summen und Mittelwertbildung
//mit diesem FB lassen sich verwirklichen:
//  - Delays, Pufferung nach dem FIFO-Prinzip
//  - Integratoren
//  - Mittelwertbildung, Dämpfungsglieder
//
//AUTOR: Stefan Maag, Dipl.-Ing. (FH) Elektrotechnik
//DATUM: 5/2003
//
//HINWEIS:
AUTHOR : 'S.Maag'
FAMILY : 'STANDARD'
VERSION : 0.1


VAR_INPUT
  WRITE : BOOL ;	//Wert in FIFO schreiben, Freigabe für Aufzeichung
  DBNr : INT ;	//Datenbaustein für FIFO
  StartAdr : INT ;	//Startadresse des ersten FIFO Eintrags im DB
  AnzahlWerte : INT ;	//Anzahl der Werte, Größe des FIFO
  FIFO_IN : INT ;	//aktueller Eingangswert der im FIFO gespeichert wird
  STARTWERT : INT ;
  RESET : BOOL ;	//FIFO zurückstellen
END_VAR
VAR_OUTPUT
  FIFO_OUT : INT ;	//Ausgangswert des FIFO
  Summe : DINT ;	//aktuelle Summe aller Werte im FIFO
  MittelWert : INT ;	//aktueller Mittelwert
  FIFO_VOLL : BOOL ;	//FIFO ist vollständig gefüllt
END_VAR
VAR
  ptrFIFO : INT ;	//Hilfsariable zum Speichern des INPUT-Zeigers
END_VAR
VAR_TEMP
  tmpDB : INT ;
  EndAdr : INT ;
  AR1 : DWORD ;
END_VAR
BEGIN
NETWORK
TITLE =RESET

      UN    #RESET;
      SPB   NE1;
      R     #FIFO_VOLL; // FIFO ist leer

      L     #AnzahlWerte;
      L     #STARTWERT;
      T     #MittelWert; // Mittelwert = Startwert
      T     #FIFO_OUT; // FIFO_OUT = Startwert
      *D    ;
      T     #Summe; // Summe=Startwert * AnzahlWerte

      L     #StartAdr; // StartAdresse im DB
      T     #ptrFIFO; // ptrFIFO_IN und

      SLD   3; // Pointer ins Bitformat
      LAR1  ;

      L     #DBNr; // DBNr
      T     #tmpDB;
      AUF   DB [#tmpDB]; // DB öffnen

// FIFO in Schleife mit Startwerten füllen
      L     #STARTWERT; // Startwert laden
      L     #AnzahlWerte; // als SchleifenZähler laden
LOOP: TAK   ; // STARTWERT in Akku1 zurück (wegen LOOP)
      T     DBW [AR1,P#0.0]; // Startwert in FIFO eintragen
      +AR1  P#2.0; // Pointer in AR1 auf nächsten Eintrag
      TAK   ; // Schleifenzähler in Akku 1
      LOOP  LOOP; // Schleifensteuerung
      BEA   ;
NE1:  NOP   0;

NETWORK
TITLE =Schreibbefehl auswerten und Baustein gegenfalls verlassen

      UN    #WRITE; // Wenn kein Schreibbefehl, dann ENDE
      BEB   ;

NETWORK
TITLE =DB öffnen und EndAdresse Datenbereich berechnen

      L     #DBNr; // DBNr
      T     #tmpDB;
      AUF   DB [#tmpDB]; // DB öffnen

      L     #AnzahlWerte; // Anzahl der Werte
      +     -1; // in Byte-Offset
      SLW   1; // konvertieren
      L     #StartAdr; // und zu Startadresse addieren
      +I    ;
      T     #EndAdr; // Endadresse Datenbereich FIFO

      L     #ptrFIFO; // FIFO Pointer
      SLD   3; // ins BitFormat
      LAR1  ; // und ins AR1
NETWORK
TITLE =FIFO voll?

      U     #FIFO_VOLL; // Wenn FIFO schon voll, dann weiter im näschten NW
      SPB   NWE;

// Eingangswert speichern und neue Summe berechnen
      L     #FIFO_IN; // Eingangswert
      T     DBW [AR1,P#0.0]; // speichern
      ITD   ;
      L     #Summe; // neue Summe
      +D    ; // berechnen und speichern
      T     #Summe;

// prüfen ob FIFO jetzt voll und Anzahl bereits enthaltener Werte berechnen
      L     #EndAdr; // Wenn ptrFIFO
      L     #ptrFIFO; // = EndAdr, dann ist FIFO voll
      ==I   ;
      S     #FIFO_VOLL; // Meldung FIFO voll
      L     #StartAdr; // ptrFIFO-StartAdr = ByteDifferenz
      -I    ;
      SRW   1; // /2 = Wortdifferenz
      +     1; // Anzahl der enthaltenen Einträge
// aktuellen Mittelwert berechnen
      L     #Summe;
      TAK   ; // Wegen Division Akkus tauschen
      /D    ; // Summe / AnzahlWerteImFIFO
      T     #MittelWert; // Mittelwert ausgeben

      SPA   PTR; // FIFO Pointer nachführen

NWE:  NOP   0;

NETWORK
TITLE =Letztwert aus FIFO entfernen, Summe und Mittelwert berechnen

      L     DBW [AR1,P#0.0]; // letzten Wert, FIFO-Out laden
      T     #FIFO_OUT; // als Ausgangswert zurückgeben
      ITD   ; // zu DINT
      L     #Summe; // Summe laden
      TAK   ; // wegen Subtraktion, Akkus tauschen
      -D    ; // FIFO-Out von Summe abziehen

      L     #FIFO_IN; // Eingangswert
      T     DBW [AR1,P#0.0]; // speichern
      ITD   ; // FIFO_IN zu DINT
      +D    ; // Summe addieren
      T     #Summe;
      L     #AnzahlWerte; // Anzahl der Werte
      /D    ; // Mittelwert berechnen
      T     #MittelWert; // Mittelwert speichern
NETWORK
TITLE =ptrFIFO auf nächsten Wert

PTR:  L     #EndAdr; // Vergleich mit Endadresse,
      L     #ptrFIFO; // Zeiger FIFO_IN auf nächsten Wert
      +     2; // +2, da ByteAdresse
      >=I   ; // solange EndAdr >, dann weitermachen
      SPB   OK; // mit neuem Pointer speichern
      L     #StartAdr; // sonst BereichsÜberlauf und weiter in StartAdr.
OK:   T     #ptrFIFO; // neuer Zeiger FIFO-IN
END_FUNCTION_BLOCK

FUNCTION_BLOCK "FIFO_INT"
TITLE =FIFO mit Summen und Mittelwertbildung
//mit diesem FC lassen sich verwirklichen:
//  - Delays, Pufferung nach dem FIFO-Prinzip
//  - Integratoren
//  - Mittelwertbildung, Dämpfungsglieder
//
//AUTOR: Stefan Maag, Dipl.-Ing. (FH) Elektrotechnik
//DATUM: 5/2003
//
//HINWEIS:
AUTHOR : 'S.Maag'
FAMILY : 'STANDARD'
VERSION : 0.1


VAR_INPUT
  DBNr : INT ;	//Datenbaustein für FIFO
  StartAdr : INT ;	//Startadresse des ersten FIFO Eintrags im DB
  AnzahlWerte : INT ;	//Anzahl der Werte, Größe des FIFO
  FIFO_IN : INT ;	//aktueller Eingangswert der im FIFO gespeichert wird
  RESET : BOOL ;	//FIFO zurückstellen
END_VAR
VAR_OUTPUT
  FIFO_OUT : INT ;	//Ausgangswert des FIFO
  Summe : DINT ;	//aktuelle Summe aller Werte im FIFO
  MittelWert : INT ;	//aktueller Mittelwert
  FIFO_VOLL : BOOL ;	//FIFO ist vollständig gefüllt
END_VAR
VAR
  ptrFIFO : INT ;	//Hilfsariable zum Speichern des INPUT-Zeigers
END_VAR
VAR_TEMP
  tmpDB : INT ;
  EndAdr : INT ;
END_VAR
BEGIN
NETWORK
TITLE =RESET

      UN    #RESET;
      SPB   WEIT;
      R     #FIFO_VOLL; // FIFO ist leer

      L     0;
      T     #Summe; // Summe löschen
      T     #MittelWert; // Mittelwert löschen
      T     #FIFO_OUT; // Ausgangswert = 0

      L     #StartAdr; // StartAdresse für
      T     #ptrFIFO; // ptrFIFO_IN und
      BEA   ;
WEIT: NOP   0;

NETWORK
TITLE =DB öffnen und EndAdresse Datenbereich berechnen

      L     #DBNr; // DBNr
      T     #tmpDB;
      AUF   DB [#tmpDB]; // DB öffnen

      L     #AnzahlWerte; // Anzahl der Werte
      +     -1; // in Byte-Offset
      SLW   1; // konvertieren
      L     #StartAdr; // und zu Startadresse addieren
      +I    ;
      T     #EndAdr; // Endadresse Datenbereich FIFO

      L     #ptrFIFO; // FIFO Pointer
      SLD   3; // ins BitFormat
      LAR1  ; // und ins AR1
NETWORK
TITLE =FIFO voll?

      U     #FIFO_VOLL; // Wenn FIFO schon voll, dann weiter im näschten NW
      SAVE  ;
      SPB   NWE;

// Eingangswert speichern und neue Summe berechnen
      L     #FIFO_IN; // Eingangswert
      T     DBW [AR1,P#0.0]; // speichern
      ITD   ;
      L     #Summe; // neue Summe
      +D    ; // berechnen und speichern
      T     #Summe;

// prüfen ob FIFO jetzt voll und Anzahl bereits enthaltener Werte berechnen
      L     #EndAdr; // Wenn ptrFIFO
      L     #ptrFIFO; // = EndAdr, dann ist FIFO voll
      ==I   ;
      S     #FIFO_VOLL; // Meldung FIFO voll
      L     #StartAdr; // ptrFIFOn-StartAdr = ByteDifferenz
      -I    ;
      SRW   1; // /2 = Wortdifferenz
      +     1; // Anzahl der enthaltenen Einträge
// aktuellen Mittelwert berechnen
      L     #Summe;
      TAK   ; // Wegen Division Akkus tauschen
      /D    ; // Summe / AnzahlWerteImFIFO
      T     #MittelWert; // Mittelwert ausgeben

      SPA   PTR; // FIFO Pointer nachführen

NWE:  NOP   0;

NETWORK
TITLE =Letztwert aus FIFO entfernen, Summe und Mittelwert berechnen

      L     DBW [AR1,P#0.0]; // letzten Wert, FIFO-Out laden
      T     #FIFO_OUT; // als Ausgangswert zurückgeben
      ITD   ; // zu DINT
      L     #Summe; // Summe laden
      TAK   ; // wegen Subtraktion, Akkus tauschen
      -D    ; // FIFO-Out von Summe abziehen

      L     #FIFO_IN; // Eingangswert
      T     DBW [AR1,P#0.0]; // speichern
      ITD   ; // FIFO_IN zu DINT
      +D    ; // Summe addieren
      T     #Summe;
      L     #AnzahlWerte; // Anzahl der Werte
      /D    ; // Mittelwert berechnen
      T     #MittelWert; // Mittelwert speichern
NETWORK
TITLE =ptrFIFO auf nächsten Wert

PTR:  L     #EndAdr; // Vergleich mit Endadresse,
      L     #ptrFIFO; // Zeiger FIFO_IN auf nächsten Wert
      +     2; // +2, da ByteAdresse
      >=I   ; // solange EndAdr >, dann weitermachen
      SPB   OK; // mit neuem Pointer speichern
      L     #StartAdr; // sonst BereichsÜberlauf und weiter in StartAdr.
OK:   T     #ptrFIFO; // neuer Zeiger FIFO-IN
END_FUNCTION_BLOCK

FUNCTION_BLOCK "m7b_FIFO_DINT_STARTWERT"
TITLE =FIFO DINT mit Startwert, Summen und Mittelwertbildung
//mit diesem FB lassen sich verwirklichen:
//  - Delays, Pufferung nach dem FIFO-Prinzip
//  - Integratoren
//  - Mittelwertbildung, Dämpfungsglieder
//
//AUTOR: Stefan Maag, Dipl.-Ing. (FH) Elektrotechnik
//DATUM: 1/2022
//
//HINWEIS:
//Entstand aus FIFO_INT_STARTWERT FB1121
AUTHOR : 'S.Maag'
FAMILY : 'STANDARD'
VERSION : 0.1


VAR_INPUT
  WRITE : BOOL ;	//Wert in FIFO schreiben, Freigabe für Aufzeichung
  BLK_DB : BLOCK_DB ;	//Datenbaustein für FIFO
  dStartAdr : DINT ;	//Startadresse des ersten FIFO Eintrags im DB
  dAnzahlWerte : INT ;	//Anzahl der Werte, Größe des FIFO
  dFIFO_IN : DINT ;	//aktueller Eingangswert der im FIFO gespeichert wird
  dStartWert : DINT ;
  RESET : BOOL ;	//FIFO zurückstellen
END_VAR
VAR_OUTPUT
  FIFO_OUT : DINT ;	//Ausgangswert des FIFO
  Summe : DINT ;	//aktuelle Summe aller Werte im FIFO
  MittelWert : DINT ;	//aktueller Mittelwert
  FIFO_VOLL : BOOL ;	//FIFO ist vollständig gefüllt
END_VAR
VAR
  ptrFIFO : DINT ;	//Hilfsariable zum Speichern des INPUT-Zeigers
END_VAR
VAR_TEMP
  dEndAdr : DINT ;
  AR1 : DWORD ;
END_VAR
BEGIN
NETWORK
TITLE =RESET

      UN    #RESET;
      SPB   NE1;
      R     #FIFO_VOLL; // FIFO ist leer

      L     #dAnzahlWerte; // Anzahl Werte [INT]
      L     #dStartWert;
      T     #MittelWert; // Mittelwert = Startwert
      T     #FIFO_OUT; // FIFO_OUT = Startwert
      *D    ;
      T     #Summe; // Summe=Startwert * AnzahlWerte

      L     #dStartAdr; // StartAdresse im DB
      T     #ptrFIFO; // ptrFIFO_IN und

      SLD   3; // Pointer ins Bitformat
      LAR1  ;

      AUF   #BLK_DB;
// FIFO in Schleife mit Startwerten füllen
      L     #dStartWert; // Startwert laden
      L     #dAnzahlWerte; // als SchleifenZähler laden
LOOP: TAK   ; // STARTWERT in Akku1 zurück (wegen LOOP)
      T     DBD [AR1,P#0.0]; // Startwert in FIFO eintragen
      +AR1  P#4.0; // Pointer in AR1 auf nächsten Eintrag
      TAK   ; // Schleifenzähler in Akku 1
      LOOP  LOOP; // Schleifensteuerung
      BEA   ;
NE1:  NOP   0;

NETWORK
TITLE =Schreibbefehl auswerten und Baustein gegenfalls verlassen

      UN    #WRITE; // Wenn kein Schreibbefehl, dann ENDE
      BEB   ;

NETWORK
TITLE =DB öffnen und EndAdresse Datenbereich berechnen

      AUF   #BLK_DB;
      L     #dAnzahlWerte; // Anzahl der Werte
      +     L#-1; // in Byte-Offset
      SLD   2; // konvertieren zu 4 Byte
      L     #dStartAdr; // und zu Startadresse addieren
      +D    ;
      T     #dEndAdr; // Endadresse Datenbereich FIFO

      L     #ptrFIFO; // FIFO Pointer
      SLD   3; // ins BitFormat
      LAR1  ; // und ins AR1
NETWORK
TITLE =FIFO voll?

      U     #FIFO_VOLL; // Wenn FIFO schon voll, dann weiter im näschten NW
      SPB   NWE;

// Eingangswert speichern und neue Summe berechnen
      L     #dFIFO_IN; // Eingangswert
      T     DBD [AR1,P#0.0]; // speichern
      L     #Summe; // neue Summe
      +R    ; // berechnen und speichern
      T     #Summe;

// prüfen ob FIFO jetzt voll und Anzahl bereits enthaltener Werte berechnen
      L     #dEndAdr; // Wenn ptrFIFO
      L     #ptrFIFO; // = EndAdr, dann ist FIFO voll
      ==D   ;
      S     #FIFO_VOLL; // Meldung FIFO voll
      L     #dStartAdr; // ptrFIFO-StartAdr = ByteDifferenz
      -D    ;
      SRD   2; // /4 = DWorddifferenz
      +     L#1; // Anzahl der enthaltenen Einträge
      DTR   ;
      L     #Summe; // aktuellen Mittelwert berechnen
      TAK   ; // Wegen Division Akkus tauschen
      /D    ; // Summe / AnzahlWerteImFIFO
      T     #MittelWert; // Mittelwert ausgeben

      SPA   PTR; // FIFO Pointer nachführen

NWE:  NOP   0;

NETWORK
TITLE =Letztwert aus FIFO entfernen, Summe und Mittelwert berechnen

      L     DBD [AR1,P#0.0]; // letzten Wert, FIFO-Out laden
      T     #FIFO_OUT; // als Ausgangswert zurückgeben
      L     #Summe; // Summe laden
      TAK   ; // wegen Subtraktion, Akkus tauschen
      -D    ; // FIFO-Out von Summe abziehen

      L     #dFIFO_IN; // Eingangswert
      T     DBD [AR1,P#0.0]; // speichern
      +D    ; // Summe addieren
      T     #Summe;
      L     #dAnzahlWerte; // Anzahl der Werte
      /D    ; // Mittelwert berechnen
      T     #MittelWert; // Mittelwert speichern
NETWORK
TITLE =ptrFIFO auf nächsten Wert

PTR:  L     #dEndAdr; // Vergleich mit Endadresse,
      L     #ptrFIFO; // Zeiger FIFO_IN auf nächsten Wert
      +     4; // +4, da ByteAdresse
      >=D   ; // solange EndAdr >, dann weitermachen
      SPB   OK; // mit neuem Pointer speichern
      L     #dStartAdr; // sonst BereichsÜberlauf und weiter in StartAdr.
OK:   T     #ptrFIFO; // neuer Zeiger FIFO-IN
END_FUNCTION_BLOCK

FUNCTION_BLOCK "m7b_FIFO_REAL_STARTWERT"
TITLE =FIFO REAL mit Startwert, Summen und Mittelwertbildung
//mit diesem FB lassen sich verwirklichen:
//  - Delays, Pufferung nach dem FIFO-Prinzip
//  - Integratoren
//  - Mittelwertbildung, Dämpfungsglieder
//
//AUTOR: Stefan Maag, Dipl.-Ing. (FH) Elektrotechnik
//DATUM: 1/2022
//
//HINWEIS:
//Entstand aus FIFO_INT_STARTWERT FB1121
AUTHOR : 'S.Maag'
FAMILY : 'STANDARD'
VERSION : 0.1


VAR_INPUT
  WRITE : BOOL ;	//Wert in FIFO schreiben, Freigabe für Aufzeichung
  BLK_DB : BLOCK_DB ;	//Datenbaustein für FIFO
  StartAdr : INT ;	//Startadresse des ersten FIFO Eintrags im DB
  iAnzahlWerte : INT ;	//Anzahl der Werte, Größe des FIFO
  FIFO_IN : REAL ;	//aktueller Eingangswert der im FIFO gespeichert wird
  STARTWERT : REAL ;
  RESET : BOOL ;	//FIFO zurückstellen
END_VAR
VAR_OUTPUT
  FIFO_OUT : REAL ;	//Ausgangswert des FIFO
  Summe : REAL ;	//aktuelle Summe aller Werte im FIFO
  MittelWert : REAL ;	//aktueller Mittelwert
  FIFO_VOLL : BOOL ;	//FIFO ist vollständig gefüllt
END_VAR
VAR
  ptrFIFO : DINT ;	//Hilfsariable zum Speichern des INPUT-Zeigers
END_VAR
VAR_TEMP
  EndAdr : DINT ;
  AR1 : DWORD ;
END_VAR
BEGIN
NETWORK
TITLE =RESET

      UN    #RESET;
      SPB   NE1;
      R     #FIFO_VOLL; // FIFO ist leer

      L     #iAnzahlWerte; // Anzahl Werte [INT]
      ITD   ;
      DTR   ;
      L     #STARTWERT;
      T     #MittelWert; // Mittelwert = Startwert
      T     #FIFO_OUT; // FIFO_OUT = Startwert
      *R    ;
      T     #Summe; // Summe=Startwert * AnzahlWerte

      L     #StartAdr; // StartAdresse im DB
      T     #ptrFIFO; // ptrFIFO_IN und

      SLD   3; // Pointer ins Bitformat
      LAR1  ;

      AUF   #BLK_DB; // DBNr
// FIFO in Schleife mit Startwerten füllen
      L     #STARTWERT; // Startwert laden
      L     #iAnzahlWerte; // als SchleifenZähler laden
LOOP: TAK   ; // STARTWERT in Akku1 zurück (wegen LOOP)
      T     DBD [AR1,P#0.0]; // Startwert in FIFO eintragen
      +AR1  P#4.0; // Pointer in AR1 auf nächsten Eintrag
      TAK   ; // Schleifenzähler in Akku 1
      LOOP  LOOP; // Schleifensteuerung
      BEA   ;
NE1:  NOP   0;

NETWORK
TITLE =Schreibbefehl auswerten und Baustein gegenfalls verlassen

      UN    #WRITE; // Wenn kein Schreibbefehl, dann ENDE
      BEB   ;

NETWORK
TITLE =DB öffnen und EndAdresse Datenbereich berechnen

      AUF   #BLK_DB; // DB öffnen
      L     #iAnzahlWerte; // Anzahl der Werte
      ITD   ;
      +     L#-1; // in Byte-Offset
      SLD   2; // konvertieren zu 4 Byte
      L     #StartAdr; // und zu Startadresse addieren
      +D    ;
      T     #EndAdr; // Endadresse Datenbereich FIFO

      L     #ptrFIFO; // FIFO Pointer
      SLD   3; // ins BitFormat
      LAR1  ; // und ins AR1
NETWORK
TITLE =FIFO voll?

      U     #FIFO_VOLL; // Wenn FIFO schon voll, dann weiter im näschten NW
      SPB   NWE;

// Eingangswert speichern und neue Summe berechnen
      L     #FIFO_IN; // Eingangswert
      T     DBD [AR1,P#0.0]; // speichern
      L     #Summe; // neue Summe
      +R    ; // berechnen und speichern
      T     #Summe;

// prüfen ob FIFO jetzt voll und Anzahl bereits enthaltener Werte berechnen
      L     #EndAdr; // Wenn ptrFIFO
      L     #ptrFIFO; // = EndAdr, dann ist FIFO voll
      ==D   ;
      S     #FIFO_VOLL; // Meldung FIFO voll
      L     #StartAdr; // ptrFIFO-StartAdr = ByteDifferenz
      -D    ;
      SRD   2; // /4 = DWorddifferenz
      +     L#1; // Anzahl der enthaltenen Einträge
      DTR   ;
      L     #Summe; // aktuellen Mittelwert berechnen
      TAK   ; // Wegen Division Akkus tauschen
      /R    ; // Summe / AnzahlWerteImFIFO
      T     #MittelWert; // Mittelwert ausgeben

      SPA   PTR; // FIFO Pointer nachführen

NWE:  NOP   0;

NETWORK
TITLE =Letztwert aus FIFO entfernen, Summe und Mittelwert berechnen

      L     DBD [AR1,P#0.0]; // letzten Wert, FIFO-Out laden
      T     #FIFO_OUT; // als Ausgangswert zurückgeben
      L     #Summe; // Summe laden
      TAK   ; // wegen Subtraktion, Akkus tauschen
      -R    ; // FIFO-Out von Summe abziehen

      L     #FIFO_IN; // Eingangswert
      T     DBD [AR1,P#0.0]; // speichern
      +R    ; // Summe addieren
      T     #Summe;
      L     #iAnzahlWerte; // Anzahl der Werte
      ITD   ;
      DTR   ;
      /R    ; // Mittelwert berechnen
      T     #MittelWert; // Mittelwert speichern
NETWORK
TITLE =ptrFIFO auf nächsten Wert

PTR:  L     #EndAdr; // Vergleich mit Endadresse,
      L     #ptrFIFO; // Zeiger FIFO_IN auf nächsten Wert
      +     4; // +4, da ByteAdresse
      >=D   ; // solange EndAdr >, dann weitermachen
      SPB   OK; // mit neuem Pointer speichern
      L     #StartAdr; // sonst BereichsÜberlauf und weiter in StartAdr.
OK:   T     #ptrFIFO; // neuer Zeiger FIFO-IN
END_FUNCTION_BLOCK

FUNCTION_BLOCK "BCD_HAND_SCHALTER"
TITLE =4 Bit BCD verzögert zu 10 digitalen Ausgängen, nur einer aktiv
//Der BCD-Wert der Eingänge BCD0 bis BCD3 werden in 10 digitale Ausgänge, von
//denen jeweils nur einer aktiv ist. Der neue BCD-Wert wird erst verzögert auf
//die Ausgänge durchgeschaltet. Dies ist nötig, wenn man einen BCD-Codierschalter
//hat und diesen als Wahlschalter zur Geräteanwahl verwendet, somit wird nicht
//bei jedem Tastendruck gleich der Steuermerker geschaltet.
//
//Zum Umschaltzeitpunkt wir der ENO-Ausgang des Bausteins für 1 Zyklus HIGH
//(Umschaltimpuls)
//
//AUTOR: Stefan Maag, Dipl.-Ing. (FH) Elektrotechnik
//DATUM: 4/2005
//
//AENDERUNGSVERMERKE:
//--------------------------------------------------------------------------------
//DATUM        NAME            AENDERUNG
//--------------------------------------------------------------------------------
//
//--------------------------------------------------------------------------------
//
//HINWEISE:
AUTHOR : 'S.Maag'
VERSION : 0.1


VAR_INPUT
  BCD0 : BOOL ;
  BCD1 : BOOL ;
  BCD2 : BOOL ;
  BCD3 : BOOL ;
  DELAY : TIME ;
END_VAR
VAR_OUTPUT
  Q0 : BOOL ;
  Q1 : BOOL ;
  Q2 : BOOL ;
  Q3 : BOOL ;
  Q4 : BOOL ;
  Q5 : BOOL ;
  Q6 : BOOL ;
  Q7 : BOOL ;
  Q8 : BOOL ;
  Q9 : BOOL ;
END_VAR
VAR
  AKT_BCD : BYTE ;
  LAST_BCD_AKTIV : BYTE ;
  LAST_BCD : BYTE ;
  CHANGE_TIME : TIME ;
  TON : "TON";
END_VAR
VAR_TEMP
  DIFF : BOOL ;
  QT : BOOL ;
  NODIFF : BOOL ;
END_VAR
BEGIN
NETWORK
TITLE =



NETWORK
TITLE =
//Wenn der Baustein als Multiinstanzaufruf verwendet wird kann nicht mit
//L DIB 0 gearbeitet werden, da es sich beim Multiinstanz-Speicher nicht
//wirklich um DIB 0 handelt, sondern mit einem Offset behaftet ist. Die
//Startadresse des Multiinstanzspeichers steht aber im Adressregister 2.
//Somit kann über die Pointer-Offsets die entsprechende Adresse geladen werden
      L     DIB [AR2,P#0.0]; // aktueller BCD Eingangswert   (lädt Byte 0 der Multiinstanz)
      L     B#16#F; // nur Bit0 bis 4
      UW    ;
      T     #AKT_BCD; // aktueller aufbereiteter BCD-WERT

      L     #AKT_BCD; // Prüfen ob der BCD
      L     #LAST_BCD_AKTIV; // Eingangswert verändert wurde
      <>I   ;
      =     #DIFF; // BCD-Wert wurde verändert

